// TIA Portal V15.1 export
// export: Created 2024-06-21T08:41:07.0870984Z, ExportSetting WithDefaults, DisplayName Totally Integrated Automation Portal, DisplayVersion V15.1 Update 5, DisplayName TIA Portal Openness, DisplayVersion V15.1 Update 5, DisplayName SINAMICS Startdrive Advanced, DisplayVersion V15.1, DisplayName G130, G150, S120, S150, SINAMICS MV, S210, DisplayVersion V15.1, DisplayName G110M, G120, G120C, G120D, G120P, DisplayVersion V15.1, DisplayName STEP 7 Professional, DisplayVersion V15.1 Update 5, DisplayName STEP 7 Safety, DisplayVersion V15.1, DisplayName WinCC Professional, DisplayVersion V15.1 Update 5, DisplayName SIMATIC Visualization Architect, DisplayVersion V15.1
FUNCTION_BLOCK "LGBBodyCounter"   // FB6602, FBD
TITLE = Body Counter Dynamic
{ S7_Optimized_Access := 'TRUE' }
AUTHOR : CSTAAL
VERSION : 0.1
// stored: AutoNumber false, IsIECCheckEnabled false, IsRetainMemResEnabled false, MemoryReserve 100, SetENOAutomatically False, UDAEnableTagReadback false
   VAR_INPUT
      I_EnableDynamicMax { ExternalAccessible := 'False'; ExternalVisible := 'False'; ExternalWritable := 'False'} : Bool;   // Dynamic Maximum Enabled
      I_MaxBody { ExternalAccessible := 'False'; ExternalVisible := 'False'; ExternalWritable := 'False'} : DInt;   // Max Amount of Bodies in the Zone
      I_DPBody { ExternalAccessible := 'False'; ExternalVisible := 'False'; ExternalWritable := 'False'} : Bool;   // DP Body Type Used in Zone
      I_ECBody { ExternalAccessible := 'False'; ExternalVisible := 'False'; ExternalWritable := 'False'} : Bool;   // EC Body Type Used in Zone
      I_ECSkid { ExternalAccessible := 'False'; ExternalVisible := 'False'; ExternalWritable := 'False'} : Bool;   // EC Skid Type Used in Zone
      I_PaintedBody { ExternalAccessible := 'False'; ExternalVisible := 'False'; ExternalWritable := 'False'} : Bool;   // Painted Body Type Used in Zone
      I_Conv1Enable { ExternalAccessible := 'False'; ExternalVisible := 'False'; ExternalWritable := 'False'} : Bool;   // Enable Conveyor 1
      I_Conv1MaxBody { ExternalAccessible := 'False'; ExternalVisible := 'False'; ExternalWritable := 'False'} : DInt;   // Max Amount of Bodies on Conveyor 1
      I_Conv1SetTrfInTrf { ExternalAccessible := 'False'; ExternalVisible := 'False'; ExternalWritable := 'False'} : Bool;   // Transfer In Set Conveyor 1
      I_Conv1SetTrfOutTrf { ExternalAccessible := 'False'; ExternalVisible := 'False'; ExternalWritable := 'False'} : Bool;   // Transfer Out Set Conveyor 1
      I_Conv1ResTrfInTrf { ExternalAccessible := 'False'; ExternalVisible := 'False'; ExternalWritable := 'False'} : Bool;   // Transfer In Reset Conveyor 1
      I_Conv1ResTrfOutTrf { ExternalAccessible := 'False'; ExternalVisible := 'False'; ExternalWritable := 'False'} : Bool;   // Transfer Out Reset Conveyor 1
      I_Conv2Enable { ExternalAccessible := 'False'; ExternalVisible := 'False'; ExternalWritable := 'False'} : Bool;   // Enable Conveyor 2
      I_Conv2MaxBody { ExternalAccessible := 'False'; ExternalVisible := 'False'; ExternalWritable := 'False'} : DInt;   // Max Amount of Bodies on Conveyor 2
      I_Conv2SetTrfInTrf { ExternalAccessible := 'False'; ExternalVisible := 'False'; ExternalWritable := 'False'} : Bool;   // Transfer In Set Conveyor 2
      I_Conv2SetTrfOutTrf { ExternalAccessible := 'False'; ExternalVisible := 'False'; ExternalWritable := 'False'} : Bool;   // Transfer Out Set Conveyor 2
      I_Conv2ResTrfInTrf { ExternalAccessible := 'False'; ExternalVisible := 'False'; ExternalWritable := 'False'} : Bool;   // Transfer In Reset Conveyor 2
      I_Conv2ResTrfOutTrf { ExternalAccessible := 'False'; ExternalVisible := 'False'; ExternalWritable := 'False'} : Bool;   // Transfer Out Reset Conveyor 2
      I_Pos1BodyPresent { ExternalAccessible := 'False'; ExternalVisible := 'False'; ExternalWritable := 'False'} : Bool;   // Position 1 Body Present
      I_Pos1RollerSetInTrf { ExternalAccessible := 'False'; ExternalVisible := 'False'; ExternalWritable := 'False'} : Bool;   // Position 1 Roller Transfer In Set
      I_Pos1RollerResInTrf { ExternalAccessible := 'False'; ExternalVisible := 'False'; ExternalWritable := 'False'} : Bool;   // Position 1 Roller Transfer In Reset
      I_Pos1CCSetInTrf { ExternalAccessible := 'False'; ExternalVisible := 'False'; ExternalWritable := 'False'} : Bool;   // Position 1 Cross Conveyor Transfer In Set
      I_Pos1CCResInTrf { ExternalAccessible := 'False'; ExternalVisible := 'False'; ExternalWritable := 'False'} : Bool;   // Position 1 Cross Conveyor Transfer In Reset
      I_Pos1RollerSetOutTrf { ExternalAccessible := 'False'; ExternalVisible := 'False'; ExternalWritable := 'False'} : Bool;   // Position 1 Roller Transfer Out Set
      I_Pos1RollerResOutTrf { ExternalAccessible := 'False'; ExternalVisible := 'False'; ExternalWritable := 'False'} : Bool;   // Position 1 Roller Transfer Out Reset
      I_Pos1CCSetOutTrf { ExternalAccessible := 'False'; ExternalVisible := 'False'; ExternalWritable := 'False'} : Bool;   // Position 1 Cross Conveyor Transfer Out Set
      I_Pos1CCResOutTrf { ExternalAccessible := 'False'; ExternalVisible := 'False'; ExternalWritable := 'False'} : Bool;   // Position 1 Cross Conveyor Transfer Out Reset
      I_Pos2BodyPresent { ExternalAccessible := 'False'; ExternalVisible := 'False'; ExternalWritable := 'False'} : Bool;   // Position 2 Body Present
      I_Pos2RollerSetInTrf { ExternalAccessible := 'False'; ExternalVisible := 'False'; ExternalWritable := 'False'} : Bool;   // Position 2 Roller Transfer In Set
      I_Pos2RollerResInTrf { ExternalAccessible := 'False'; ExternalVisible := 'False'; ExternalWritable := 'False'} : Bool;   // Position 2 Roller Transfer In Reset
      I_Pos2CCSetInTrf { ExternalAccessible := 'False'; ExternalVisible := 'False'; ExternalWritable := 'False'} : Bool;   // Position 2 Cross Conveyor Transfer In Set
      I_Pos2CCResInTrf { ExternalAccessible := 'False'; ExternalVisible := 'False'; ExternalWritable := 'False'} : Bool;   // Position 2 Cross Conveyor Transfer In Reset
      I_Pos2RollerSetOutTrf { ExternalAccessible := 'False'; ExternalVisible := 'False'; ExternalWritable := 'False'} : Bool;   // Position 2 Roller Transfer Out Set
      I_Pos2RollerResOutTrf { ExternalAccessible := 'False'; ExternalVisible := 'False'; ExternalWritable := 'False'} : Bool;   // Position 2 Roller Transfer Out Reset
      I_Pos2CCSetOutTrf { ExternalAccessible := 'False'; ExternalVisible := 'False'; ExternalWritable := 'False'} : Bool;   // Position 2 Cross Conveyor Transfer Out Set
      I_Pos2CCResOutTrf { ExternalAccessible := 'False'; ExternalVisible := 'False'; ExternalWritable := 'False'} : Bool;   // Position 2 Cross Conveyor Transfer Out Reset
      I_Pos3BodyPresent { ExternalAccessible := 'False'; ExternalVisible := 'False'; ExternalWritable := 'False'} : Bool;   // Position 3 Body Present
      I_Pos3RollerSetInTrf { ExternalAccessible := 'False'; ExternalVisible := 'False'; ExternalWritable := 'False'} : Bool;   // Position 3 Roller Transfer In Set
      I_Pos3RollerResInTrf { ExternalAccessible := 'False'; ExternalVisible := 'False'; ExternalWritable := 'False'} : Bool;   // Position 3 Roller Transfer In Reset
      I_Pos3CCSetInTrf { ExternalAccessible := 'False'; ExternalVisible := 'False'; ExternalWritable := 'False'} : Bool;   // Position 3 Cross Conveyor Transfer In Set
      I_Pos3CCResInTrf { ExternalAccessible := 'False'; ExternalVisible := 'False'; ExternalWritable := 'False'} : Bool;   // Position 3 Cross Conveyor Transfer In Reset
      I_Pos3RollerSetOutTrf { ExternalAccessible := 'False'; ExternalVisible := 'False'; ExternalWritable := 'False'} : Bool;   // Position 3 Roller Transfer Out Set
      I_Pos3RollerResOutTrf { ExternalAccessible := 'False'; ExternalVisible := 'False'; ExternalWritable := 'False'} : Bool;   // Position 3 Roller Transfer Out Reset
      I_Pos3CCSetOutTrf { ExternalAccessible := 'False'; ExternalVisible := 'False'; ExternalWritable := 'False'} : Bool;   // Position 3 Cross Conveyor Transfer Out Set
      I_Pos3CCResOutTrf { ExternalAccessible := 'False'; ExternalVisible := 'False'; ExternalWritable := 'False'} : Bool;   // Position 3 Cross Conveyor Transfer Out Reset
      I_Pos4BodyPresent { ExternalAccessible := 'False'; ExternalVisible := 'False'; ExternalWritable := 'False'} : Bool;   // Position 4 Body Present
      I_Pos4RollerSetInTrf { ExternalAccessible := 'False'; ExternalVisible := 'False'; ExternalWritable := 'False'} : Bool;   // Position 4 Roller Transfer In Set
      I_Pos4RollerResInTrf { ExternalAccessible := 'False'; ExternalVisible := 'False'; ExternalWritable := 'False'} : Bool;   // Position 4 Roller Transfer In Reset
      I_Pos4CCSetInTrf { ExternalAccessible := 'False'; ExternalVisible := 'False'; ExternalWritable := 'False'} : Bool;   // Position 4 Cross Conveyor Transfer In Set
      I_Pos4CCResInTrf { ExternalAccessible := 'False'; ExternalVisible := 'False'; ExternalWritable := 'False'} : Bool;   // Position 4 Cross Conveyor Transfer In Reset
      I_Pos4RollerSetOutTrf { ExternalAccessible := 'False'; ExternalVisible := 'False'; ExternalWritable := 'False'} : Bool;   // Position 4 Roller Transfer Out Set
      I_Pos4RollerResOutTrf { ExternalAccessible := 'False'; ExternalVisible := 'False'; ExternalWritable := 'False'} : Bool;   // Position 4 Roller Transfer Out Reset
      I_Pos4CCSetOutTrf { ExternalAccessible := 'False'; ExternalVisible := 'False'; ExternalWritable := 'False'} : Bool;   // Position 4 Cross Conveyor Transfer Out Set
      I_Pos4CCResOutTrf { ExternalAccessible := 'False'; ExternalVisible := 'False'; ExternalWritable := 'False'} : Bool;   // Position 4 Cross Conveyor Transfer Out Reset
      I_Pos5BodyPresent { ExternalAccessible := 'False'; ExternalVisible := 'False'; ExternalWritable := 'False'} : Bool;   // Position 5 Body Present
      I_Pos5RollerSetInTrf { ExternalAccessible := 'False'; ExternalVisible := 'False'; ExternalWritable := 'False'} : Bool;   // Position 5 Roller Transfer In Set
      I_Pos5RollerResInTrf { ExternalAccessible := 'False'; ExternalVisible := 'False'; ExternalWritable := 'False'} : Bool;   // Position 5 Roller Transfer In Reset
      I_Pos5CCSetInTrf { ExternalAccessible := 'False'; ExternalVisible := 'False'; ExternalWritable := 'False'} : Bool;   // Position 5 Cross Conveyor Transfer In Set
      I_Pos5CCResInTrf { ExternalAccessible := 'False'; ExternalVisible := 'False'; ExternalWritable := 'False'} : Bool;   // Position 5 Cross Conveyor Transfer In Reset
      I_Pos5RollerSetOutTrf { ExternalAccessible := 'False'; ExternalVisible := 'False'; ExternalWritable := 'False'} : Bool;   // Position 5 Roller Transfer Out Set
      I_Pos5RollerResOutTrf { ExternalAccessible := 'False'; ExternalVisible := 'False'; ExternalWritable := 'False'} : Bool;   // Position 5 Roller Transfer Out Reset
      I_Pos5CCSetOutTrf { ExternalAccessible := 'False'; ExternalVisible := 'False'; ExternalWritable := 'False'} : Bool;   // Position 5 Cross Conveyor Transfer Out Set
      I_Pos5CCResOutTrf { ExternalAccessible := 'False'; ExternalVisible := 'False'; ExternalWritable := 'False'} : Bool;   // Position 5 Cross Conveyor Transfer Out Reset
      I_Pos6BodyPresent { ExternalAccessible := 'False'; ExternalVisible := 'False'; ExternalWritable := 'False'} : Bool;   // Position 6 Body Present
      I_Pos6RollerSetInTrf { ExternalAccessible := 'False'; ExternalVisible := 'False'; ExternalWritable := 'False'} : Bool;   // Position 6 Roller Transfer In Set
      I_Pos6RollerResInTrf { ExternalAccessible := 'False'; ExternalVisible := 'False'; ExternalWritable := 'False'} : Bool;   // Position 6 Roller Transfer In Reset
      I_Pos6CCSetInTrf { ExternalAccessible := 'False'; ExternalVisible := 'False'; ExternalWritable := 'False'} : Bool;   // Position 6 Cross Conveyor Transfer In Set
      I_Pos6CCResInTrf { ExternalAccessible := 'False'; ExternalVisible := 'False'; ExternalWritable := 'False'} : Bool;   // Position 6 Cross Conveyor Transfer In Reset
      I_Pos6RollerSetOutTrf { ExternalAccessible := 'False'; ExternalVisible := 'False'; ExternalWritable := 'False'} : Bool;   // Position 6 Roller Transfer Out Set
      I_Pos6RollerResOutTrf { ExternalAccessible := 'False'; ExternalVisible := 'False'; ExternalWritable := 'False'} : Bool;   // Position 6 Roller Transfer Out Reset
      I_Pos6CCSetOutTrf { ExternalAccessible := 'False'; ExternalVisible := 'False'; ExternalWritable := 'False'} : Bool;   // Position 6 Cross Conveyor Transfer Out Set
      I_Pos6CCResOutTrf { ExternalAccessible := 'False'; ExternalVisible := 'False'; ExternalWritable := 'False'} : Bool;   // Position 6 Cross Conveyor Transfer Out Reset
      I_Pos7BodyPresent { ExternalAccessible := 'False'; ExternalVisible := 'False'; ExternalWritable := 'False'} : Bool;   // Position 7 Body Present
      I_Pos7RollerSetInTrf { ExternalAccessible := 'False'; ExternalVisible := 'False'; ExternalWritable := 'False'} : Bool;   // Position 7 Roller Transfer In Set
      I_Pos7RollerResInTrf { ExternalAccessible := 'False'; ExternalVisible := 'False'; ExternalWritable := 'False'} : Bool;   // Position 7 Roller Transfer In Reset
      I_Pos7CCSetInTrf { ExternalAccessible := 'False'; ExternalVisible := 'False'; ExternalWritable := 'False'} : Bool;   // Position 7 Cross Conveyor Transfer In Set
      I_Pos7CCResInTrf { ExternalAccessible := 'False'; ExternalVisible := 'False'; ExternalWritable := 'False'} : Bool;   // Position 7 Cross Conveyor Transfer In Reset
      I_Pos7RollerSetOutTrf { ExternalAccessible := 'False'; ExternalVisible := 'False'; ExternalWritable := 'False'} : Bool;   // Position 7 Roller Transfer Out Set
      I_Pos7RollerResOutTrf { ExternalAccessible := 'False'; ExternalVisible := 'False'; ExternalWritable := 'False'} : Bool;   // Position 7 Roller Transfer Out Reset
      I_Pos7CCSetOutTrf { ExternalAccessible := 'False'; ExternalVisible := 'False'; ExternalWritable := 'False'} : Bool;   // Position 7 Cross Conveyor Transfer Out Set
      I_Pos7CCResOutTrf { ExternalAccessible := 'False'; ExternalVisible := 'False'; ExternalWritable := 'False'} : Bool;   // Position 7 Cross Conveyor Transfer Out Reset
      I_Pos8BodyPresent { ExternalAccessible := 'False'; ExternalVisible := 'False'; ExternalWritable := 'False'} : Bool;   // Position 8 Body Present
      I_Pos8RollerSetInTrf { ExternalAccessible := 'False'; ExternalVisible := 'False'; ExternalWritable := 'False'} : Bool;   // Position 8 Roller Transfer In Set
      I_Pos8RollerResInTrf { ExternalAccessible := 'False'; ExternalVisible := 'False'; ExternalWritable := 'False'} : Bool;   // Position 8 Roller Transfer In Reset
      I_Pos8CCSetInTrf { ExternalAccessible := 'False'; ExternalVisible := 'False'; ExternalWritable := 'False'} : Bool;   // Position 8 Cross Conveyor Transfer In Set
      I_Pos8CCResInTrf { ExternalAccessible := 'False'; ExternalVisible := 'False'; ExternalWritable := 'False'} : Bool;   // Position 8 Cross Conveyor Transfer In Reset
      I_Pos8RollerSetOutTrf { ExternalAccessible := 'False'; ExternalVisible := 'False'; ExternalWritable := 'False'} : Bool;   // Position 8 Roller Transfer Out Set
      I_Pos8RollerResOutTrf { ExternalAccessible := 'False'; ExternalVisible := 'False'; ExternalWritable := 'False'} : Bool;   // Position 8 Roller Transfer Out Reset
      I_Pos8CCSetOutTrf { ExternalAccessible := 'False'; ExternalVisible := 'False'; ExternalWritable := 'False'} : Bool;   // Position 8 Cross Conveyor Transfer Out Set
      I_Pos8CCResOutTrf { ExternalAccessible := 'False'; ExternalVisible := 'False'; ExternalWritable := 'False'} : Bool;   // Position 8 Cross Conveyor Transfer Out Reset
      I_Pos9BodyPresent { ExternalAccessible := 'False'; ExternalVisible := 'False'; ExternalWritable := 'False'} : Bool;   // Position 9 Body Present
      I_Pos9RollerSetInTrf { ExternalAccessible := 'False'; ExternalVisible := 'False'; ExternalWritable := 'False'} : Bool;   // Position 9 Roller Transfer In Set
      I_Pos9RollerResInTrf { ExternalAccessible := 'False'; ExternalVisible := 'False'; ExternalWritable := 'False'} : Bool;   // Position 9 Roller Transfer In Reset
      I_Pos9CCSetInTrf { ExternalAccessible := 'False'; ExternalVisible := 'False'; ExternalWritable := 'False'} : Bool;   // Position 9 Cross Conveyor Transfer In Set
      I_Pos9CCResInTrf { ExternalAccessible := 'False'; ExternalVisible := 'False'; ExternalWritable := 'False'} : Bool;   // Position 9 Cross Conveyor Transfer In Reset
      I_Pos9RollerSetOutTrf { ExternalAccessible := 'False'; ExternalVisible := 'False'; ExternalWritable := 'False'} : Bool;   // Position 9 Roller Transfer Out Set
      I_Pos9RollerResOutTrf { ExternalAccessible := 'False'; ExternalVisible := 'False'; ExternalWritable := 'False'} : Bool;   // Position 9 Roller Transfer Out Reset
      I_Pos9CCSetOutTrf { ExternalAccessible := 'False'; ExternalVisible := 'False'; ExternalWritable := 'False'} : Bool;   // Position 9 Cross Conveyor Transfer Out Set
      I_Pos9CCResOutTrf { ExternalAccessible := 'False'; ExternalVisible := 'False'; ExternalWritable := 'False'} : Bool;   // Position 9 Cross Conveyor Transfer Out Reset
      I_Pos10BodyPresent { ExternalAccessible := 'False'; ExternalVisible := 'False'; ExternalWritable := 'False'} : Bool;   // Position 10 Body Present
      I_Pos10RollerSetInTrf { ExternalAccessible := 'False'; ExternalVisible := 'False'; ExternalWritable := 'False'} : Bool;   // Position 10 Roller Transfer In Set
      I_Pos10RollerResInTrf { ExternalAccessible := 'False'; ExternalVisible := 'False'; ExternalWritable := 'False'} : Bool;   // Position 10 Roller Transfer In Reset
      I_Pos10CCSetInTrf { ExternalAccessible := 'False'; ExternalVisible := 'False'; ExternalWritable := 'False'} : Bool;   // Position 10 Cross Conveyor Transfer In Set
      I_Pos10CCResInTrf { ExternalAccessible := 'False'; ExternalVisible := 'False'; ExternalWritable := 'False'} : Bool;   // Position 10 Cross Conveyor Transfer In Reset
      I_Pos10RollerSetOutTrf { ExternalAccessible := 'False'; ExternalVisible := 'False'; ExternalWritable := 'False'} : Bool;   // Position 10 Roller Transfer Out Set
      I_Pos10RollerResOutTrf { ExternalAccessible := 'False'; ExternalVisible := 'False'; ExternalWritable := 'False'} : Bool;   // Position 10 Roller Transfer Out Reset
      I_Pos10CCSetOutTrf { ExternalAccessible := 'False'; ExternalVisible := 'False'; ExternalWritable := 'False'} : Bool;   // Position 10 Cross Conveyor Transfer Out Set
      I_Pos10CCResOutTrf { ExternalAccessible := 'False'; ExternalVisible := 'False'; ExternalWritable := 'False'} : Bool;   // Position 10 Cross Conveyor Transfer Out Reset
      I_Pos11BodyPresent { ExternalAccessible := 'False'; ExternalVisible := 'False'; ExternalWritable := 'False'} : Bool;   // Position 11 Body Present
      I_Pos11RollerSetInTrf { ExternalAccessible := 'False'; ExternalVisible := 'False'; ExternalWritable := 'False'} : Bool;   // Position 11 Roller Transfer In Set
      I_Pos11RollerResInTrf { ExternalAccessible := 'False'; ExternalVisible := 'False'; ExternalWritable := 'False'} : Bool;   // Position 11 Roller Transfer In Reset
      I_Pos11CCSetInTrf { ExternalAccessible := 'False'; ExternalVisible := 'False'; ExternalWritable := 'False'} : Bool;   // Position 11 Cross Conveyor Transfer In Set
      I_Pos11CCResInTrf { ExternalAccessible := 'False'; ExternalVisible := 'False'; ExternalWritable := 'False'} : Bool;   // Position 11 Cross Conveyor Transfer In Reset
      I_Pos11RollerSetOutTrf { ExternalAccessible := 'False'; ExternalVisible := 'False'; ExternalWritable := 'False'} : Bool;   // Position 11 Roller Transfer Out Set
      I_Pos11RollerResOutTrf { ExternalAccessible := 'False'; ExternalVisible := 'False'; ExternalWritable := 'False'} : Bool;   // Position 11 Roller Transfer Out Reset
      I_Pos11CCSetOutTrf { ExternalAccessible := 'False'; ExternalVisible := 'False'; ExternalWritable := 'False'} : Bool;   // Position 11 Cross Conveyor Transfer Out Set
      I_Pos11CCResOutTrf { ExternalAccessible := 'False'; ExternalVisible := 'False'; ExternalWritable := 'False'} : Bool;   // Position 11 Cross Conveyor Transfer Out Reset
      I_Pos12BodyPresent { ExternalAccessible := 'False'; ExternalVisible := 'False'; ExternalWritable := 'False'} : Bool;   // Position 12 Body Present
      I_Pos12RollerSetInTrf { ExternalAccessible := 'False'; ExternalVisible := 'False'; ExternalWritable := 'False'} : Bool;   // Position 12 Roller Transfer In Set
      I_Pos12RollerResInTrf { ExternalAccessible := 'False'; ExternalVisible := 'False'; ExternalWritable := 'False'} : Bool;   // Position 12 Roller Transfer In Reset
      I_Pos12CCSetInTrf { ExternalAccessible := 'False'; ExternalVisible := 'False'; ExternalWritable := 'False'} : Bool;   // Position 12 Cross Conveyor Transfer In Set
      I_Pos12CCResInTrf { ExternalAccessible := 'False'; ExternalVisible := 'False'; ExternalWritable := 'False'} : Bool;   // Position 12 Cross Conveyor Transfer In Reset
      I_Pos12RollerSetOutTrf { ExternalAccessible := 'False'; ExternalVisible := 'False'; ExternalWritable := 'False'} : Bool;   // Position 12 Roller Transfer Out Set
      I_Pos12RollerResOutTrf { ExternalAccessible := 'False'; ExternalVisible := 'False'; ExternalWritable := 'False'} : Bool;   // Position 12 Roller Transfer Out Reset
      I_Pos12CCSetOutTrf { ExternalAccessible := 'False'; ExternalVisible := 'False'; ExternalWritable := 'False'} : Bool;   // Position 12 Cross Conveyor Transfer Out Set
      I_Pos12CCResOutTrf { ExternalAccessible := 'False'; ExternalVisible := 'False'; ExternalWritable := 'False'} : Bool;   // Position 12 Cross Conveyor Transfer Out Reset
      I_Pos13BodyPresent { ExternalAccessible := 'False'; ExternalVisible := 'False'; ExternalWritable := 'False'} : Bool;   // Position 13 Body Present
      I_Pos13RollerSetInTrf { ExternalAccessible := 'False'; ExternalVisible := 'False'; ExternalWritable := 'False'} : Bool;   // Position 13 Roller Transfer In Set
      I_Pos13RollerResInTrf { ExternalAccessible := 'False'; ExternalVisible := 'False'; ExternalWritable := 'False'} : Bool;   // Position 13 Roller Transfer In Reset
      I_Pos13CCSetInTrf { ExternalAccessible := 'False'; ExternalVisible := 'False'; ExternalWritable := 'False'} : Bool;   // Position 13 Cross Conveyor Transfer In Set
      I_Pos13CCResInTrf { ExternalAccessible := 'False'; ExternalVisible := 'False'; ExternalWritable := 'False'} : Bool;   // Position 13 Cross Conveyor Transfer In Reset
      I_Pos13RollerSetOutTrf { ExternalAccessible := 'False'; ExternalVisible := 'False'; ExternalWritable := 'False'} : Bool;   // Position 13 Roller Transfer Out Set
      I_Pos13RollerResOutTrf { ExternalAccessible := 'False'; ExternalVisible := 'False'; ExternalWritable := 'False'} : Bool;   // Position 13 Roller Transfer Out Reset
      I_Pos13CCSetOutTrf { ExternalAccessible := 'False'; ExternalVisible := 'False'; ExternalWritable := 'False'} : Bool;   // Position 13 Cross Conveyor Transfer Out Set
      I_Pos13CCResOutTrf { ExternalAccessible := 'False'; ExternalVisible := 'False'; ExternalWritable := 'False'} : Bool;   // Position 13 Cross Conveyor Transfer Out Reset
      I_Pos14BodyPresent { ExternalAccessible := 'False'; ExternalVisible := 'False'; ExternalWritable := 'False'} : Bool;   // Position 14 Body Present
      I_Pos14RollerSetInTrf { ExternalAccessible := 'False'; ExternalVisible := 'False'; ExternalWritable := 'False'} : Bool;   // Position 14 Roller Transfer In Set
      I_Pos14RollerResInTrf { ExternalAccessible := 'False'; ExternalVisible := 'False'; ExternalWritable := 'False'} : Bool;   // Position 14 Roller Transfer In Reset
      I_Pos14CCSetInTrf { ExternalAccessible := 'False'; ExternalVisible := 'False'; ExternalWritable := 'False'} : Bool;   // Position 14 Cross Conveyor Transfer In Set
      I_Pos14CCResInTrf { ExternalAccessible := 'False'; ExternalVisible := 'False'; ExternalWritable := 'False'} : Bool;   // Position 14 Cross Conveyor Transfer In Reset
      I_Pos14RollerSetOutTrf { ExternalAccessible := 'False'; ExternalVisible := 'False'; ExternalWritable := 'False'} : Bool;   // Position 14 Roller Transfer Out Set
      I_Pos14RollerResOutTrf { ExternalAccessible := 'False'; ExternalVisible := 'False'; ExternalWritable := 'False'} : Bool;   // Position 14 Roller Transfer Out Reset
      I_Pos14CCSetOutTrf { ExternalAccessible := 'False'; ExternalVisible := 'False'; ExternalWritable := 'False'} : Bool;   // Position 14 Cross Conveyor Transfer Out Set
      I_Pos14CCResOutTrf { ExternalAccessible := 'False'; ExternalVisible := 'False'; ExternalWritable := 'False'} : Bool;   // Position 14 Cross Conveyor Transfer Out Reset
      I_Pos15BodyPresent { ExternalAccessible := 'False'; ExternalVisible := 'False'; ExternalWritable := 'False'} : Bool;   // Position 15 Body Present
      I_Pos15RollerSetInTrf { ExternalAccessible := 'False'; ExternalVisible := 'False'; ExternalWritable := 'False'} : Bool;   // Position 15 Roller Transfer In Set
      I_Pos15RollerResInTrf { ExternalAccessible := 'False'; ExternalVisible := 'False'; ExternalWritable := 'False'} : Bool;   // Position 15 Roller Transfer In Reset
      I_Pos15CCSetInTrf { ExternalAccessible := 'False'; ExternalVisible := 'False'; ExternalWritable := 'False'} : Bool;   // Position 15 Cross Conveyor Transfer In Set
      I_Pos15CCResInTrf { ExternalAccessible := 'False'; ExternalVisible := 'False'; ExternalWritable := 'False'} : Bool;   // Position 15 Cross Conveyor Transfer In Reset
      I_Pos15RollerSetOutTrf { ExternalAccessible := 'False'; ExternalVisible := 'False'; ExternalWritable := 'False'} : Bool;   // Position 15 Roller Transfer Out Set
      I_Pos15RollerResOutTrf { ExternalAccessible := 'False'; ExternalVisible := 'False'; ExternalWritable := 'False'} : Bool;   // Position 15 Roller Transfer Out Reset
      I_Pos15CCSetOutTrf { ExternalAccessible := 'False'; ExternalVisible := 'False'; ExternalWritable := 'False'} : Bool;   // Position 15 Cross Conveyor Transfer Out Set
      I_Pos15CCResOutTrf { ExternalAccessible := 'False'; ExternalVisible := 'False'; ExternalWritable := 'False'} : Bool;   // Position 15 Cross Conveyor Transfer Out Reset
      I_Pos16BodyPresent { ExternalAccessible := 'False'; ExternalVisible := 'False'; ExternalWritable := 'False'} : Bool;   // Position 16 Body Present
      I_Pos16RollerSetInTrf { ExternalAccessible := 'False'; ExternalVisible := 'False'; ExternalWritable := 'False'} : Bool;   // Position 16 Roller Transfer In Set
      I_Pos16RollerResInTrf { ExternalAccessible := 'False'; ExternalVisible := 'False'; ExternalWritable := 'False'} : Bool;   // Position 16 Roller Transfer In Reset
      I_Pos16CCSetInTrf { ExternalAccessible := 'False'; ExternalVisible := 'False'; ExternalWritable := 'False'} : Bool;   // Position 16 Cross Conveyor Transfer In Set
      I_Pos16CCResInTrf { ExternalAccessible := 'False'; ExternalVisible := 'False'; ExternalWritable := 'False'} : Bool;   // Position 16 Cross Conveyor Transfer In Reset
      I_Pos16RollerSetOutTrf { ExternalAccessible := 'False'; ExternalVisible := 'False'; ExternalWritable := 'False'} : Bool;   // Position 16 Roller Transfer Out Set
      I_Pos16RollerResOutTrf { ExternalAccessible := 'False'; ExternalVisible := 'False'; ExternalWritable := 'False'} : Bool;   // Position 16 Roller Transfer Out Reset
      I_Pos16CCSetOutTrf { ExternalAccessible := 'False'; ExternalVisible := 'False'; ExternalWritable := 'False'} : Bool;   // Position 16 Cross Conveyor Transfer Out Set
      I_Pos16CCResOutTrf { ExternalAccessible := 'False'; ExternalVisible := 'False'; ExternalWritable := 'False'} : Bool;   // Position 16 Cross Conveyor Transfer Out Reset
      I_Pos17BodyPresent { ExternalAccessible := 'False'; ExternalVisible := 'False'; ExternalWritable := 'False'} : Bool;   // Position 17 Body Present
      I_Pos17RollerSetInTrf { ExternalAccessible := 'False'; ExternalVisible := 'False'; ExternalWritable := 'False'} : Bool;   // Position 17 Roller Transfer In Set
      I_Pos17RollerResInTrf { ExternalAccessible := 'False'; ExternalVisible := 'False'; ExternalWritable := 'False'} : Bool;   // Position 17 Roller Transfer In Reset
      I_Pos17CCSetInTrf { ExternalAccessible := 'False'; ExternalVisible := 'False'; ExternalWritable := 'False'} : Bool;   // Position 17 Cross Conveyor Transfer In Set
      I_Pos17CCResInTrf { ExternalAccessible := 'False'; ExternalVisible := 'False'; ExternalWritable := 'False'} : Bool;   // Position 17 Cross Conveyor Transfer In Reset
      I_Pos17RollerSetOutTrf { ExternalAccessible := 'False'; ExternalVisible := 'False'; ExternalWritable := 'False'} : Bool;   // Position 17 Roller Transfer Out Set
      I_Pos17RollerResOutTrf { ExternalAccessible := 'False'; ExternalVisible := 'False'; ExternalWritable := 'False'} : Bool;   // Position 17 Roller Transfer Out Reset
      I_Pos17CCSetOutTrf { ExternalAccessible := 'False'; ExternalVisible := 'False'; ExternalWritable := 'False'} : Bool;   // Position 17 Cross Conveyor Transfer Out Set
      I_Pos17CCResOutTrf { ExternalAccessible := 'False'; ExternalVisible := 'False'; ExternalWritable := 'False'} : Bool;   // Position 17 Cross Conveyor Transfer Out Reset
      I_Pos18BodyPresent { ExternalAccessible := 'False'; ExternalVisible := 'False'; ExternalWritable := 'False'} : Bool;   // Position 18 Body Present
      I_Pos18RollerSetInTrf { ExternalAccessible := 'False'; ExternalVisible := 'False'; ExternalWritable := 'False'} : Bool;   // Position 18 Roller Transfer In Set
      I_Pos18RollerResInTrf { ExternalAccessible := 'False'; ExternalVisible := 'False'; ExternalWritable := 'False'} : Bool;   // Position 18 Roller Transfer In Reset
      I_Pos18CCSetInTrf { ExternalAccessible := 'False'; ExternalVisible := 'False'; ExternalWritable := 'False'} : Bool;   // Position 18 Cross Conveyor Transfer In Set
      I_Pos18CCResInTrf { ExternalAccessible := 'False'; ExternalVisible := 'False'; ExternalWritable := 'False'} : Bool;   // Position 18 Cross Conveyor Transfer In Reset
      I_Pos18RollerSetOutTrf { ExternalAccessible := 'False'; ExternalVisible := 'False'; ExternalWritable := 'False'} : Bool;   // Position 18 Roller Transfer Out Set
      I_Pos18RollerResOutTrf { ExternalAccessible := 'False'; ExternalVisible := 'False'; ExternalWritable := 'False'} : Bool;   // Position 18 Roller Transfer Out Reset
      I_Pos18CCSetOutTrf { ExternalAccessible := 'False'; ExternalVisible := 'False'; ExternalWritable := 'False'} : Bool;   // Position 18 Cross Conveyor Transfer Out Set
      I_Pos18CCResOutTrf { ExternalAccessible := 'False'; ExternalVisible := 'False'; ExternalWritable := 'False'} : Bool;   // Position 18 Cross Conveyor Transfer Out Reset
      I_Pos19BodyPresent { ExternalAccessible := 'False'; ExternalVisible := 'False'; ExternalWritable := 'False'} : Bool;   // Position 19 Body Present
      I_Pos19RollerSetInTrf { ExternalAccessible := 'False'; ExternalVisible := 'False'; ExternalWritable := 'False'} : Bool;   // Position 19 Roller Transfer In Set
      I_Pos19RollerResInTrf { ExternalAccessible := 'False'; ExternalVisible := 'False'; ExternalWritable := 'False'} : Bool;   // Position 19 Roller Transfer In Reset
      I_Pos19CCSetInTrf { ExternalAccessible := 'False'; ExternalVisible := 'False'; ExternalWritable := 'False'} : Bool;   // Position 19 Cross Conveyor Transfer In Set
      I_Pos19CCResInTrf { ExternalAccessible := 'False'; ExternalVisible := 'False'; ExternalWritable := 'False'} : Bool;   // Position 19 Cross Conveyor Transfer In Reset
      I_Pos19RollerSetOutTrf { ExternalAccessible := 'False'; ExternalVisible := 'False'; ExternalWritable := 'False'} : Bool;   // Position 19 Roller Transfer Out Set
      I_Pos19RollerResOutTrf { ExternalAccessible := 'False'; ExternalVisible := 'False'; ExternalWritable := 'False'} : Bool;   // Position 19 Roller Transfer Out Reset
      I_Pos19CCSetOutTrf { ExternalAccessible := 'False'; ExternalVisible := 'False'; ExternalWritable := 'False'} : Bool;   // Position 19 Cross Conveyor Transfer Out Set
      I_Pos19CCResOutTrf { ExternalAccessible := 'False'; ExternalVisible := 'False'; ExternalWritable := 'False'} : Bool;   // Position 19 Cross Conveyor Transfer Out Reset
      I_Pos20BodyPresent { ExternalAccessible := 'False'; ExternalVisible := 'False'; ExternalWritable := 'False'} : Bool;   // Position 20 Body Present
      I_Pos20RollerSetInTrf { ExternalAccessible := 'False'; ExternalVisible := 'False'; ExternalWritable := 'False'} : Bool;   // Position 20 Roller Transfer In Set
      I_Pos20RollerResInTrf { ExternalAccessible := 'False'; ExternalVisible := 'False'; ExternalWritable := 'False'} : Bool;   // Position 20 Roller Transfer In Reset
      I_Pos20CCSetInTrf { ExternalAccessible := 'False'; ExternalVisible := 'False'; ExternalWritable := 'False'} : Bool;   // Position 20 Cross Conveyor Transfer In Set
      I_Pos20CCResInTrf { ExternalAccessible := 'False'; ExternalVisible := 'False'; ExternalWritable := 'False'} : Bool;   // Position 20 Cross Conveyor Transfer In Reset
      I_Pos20RollerSetOutTrf { ExternalAccessible := 'False'; ExternalVisible := 'False'; ExternalWritable := 'False'} : Bool;   // Position 20 Roller Transfer Out Set
      I_Pos20RollerResOutTrf { ExternalAccessible := 'False'; ExternalVisible := 'False'; ExternalWritable := 'False'} : Bool;   // Position 20 Roller Transfer Out Reset
      I_Pos20CCSetOutTrf { ExternalAccessible := 'False'; ExternalVisible := 'False'; ExternalWritable := 'False'} : Bool;   // Position 20 Cross Conveyor Transfer Out Set
      I_Pos20CCResOutTrf { ExternalAccessible := 'False'; ExternalVisible := 'False'; ExternalWritable := 'False'} : Bool;   // Position 20 Cross Conveyor Transfer Out Reset
      I_Pos21BodyPresent { ExternalAccessible := 'False'; ExternalVisible := 'False'; ExternalWritable := 'False'} : Bool;   // Position 21 Body Present
      I_Pos21CCResOutTrf { ExternalAccessible := 'False'; ExternalVisible := 'False'; ExternalWritable := 'False'} : Bool;   // Position 21 Cross Conveyor Transfer Out Reset
      I_Pos21RollerSetInTrf { ExternalAccessible := 'False'; ExternalVisible := 'False'; ExternalWritable := 'False'} : Bool;   // Position 21 Roller Transfer In Set
      I_Pos21RollerResInTrf { ExternalAccessible := 'False'; ExternalVisible := 'False'; ExternalWritable := 'False'} : Bool;   // Position 21 Roller Transfer In Reset
      I_Pos21CCResInTrf { ExternalAccessible := 'False'; ExternalVisible := 'False'; ExternalWritable := 'False'} : Bool;   // Position 21 Cross Conveyor Transfer In Reset
      I_Pos21CCSetInTrf { ExternalAccessible := 'False'; ExternalVisible := 'False'; ExternalWritable := 'False'} : Bool;   // Position 21 Cross Conveyor Transfer In Set
      I_Pos21RollerSetOutTrf { ExternalAccessible := 'False'; ExternalVisible := 'False'; ExternalWritable := 'False'} : Bool;   // Position 21 Roller Transfer Out Set
      I_Pos21RollerResOutTrf { ExternalAccessible := 'False'; ExternalVisible := 'False'; ExternalWritable := 'False'} : Bool;   // Position 21 Roller Transfer Out Reset
      I_Pos21CCSetOutTrf { ExternalAccessible := 'False'; ExternalVisible := 'False'; ExternalWritable := 'False'} : Bool;   // Position 21 Cross Conveyor Transfer Out Set
      I_Pos22BodyPresent { ExternalAccessible := 'False'; ExternalVisible := 'False'; ExternalWritable := 'False'} : Bool;   // Position 22 Body Present
      I_Pos22CCResOutTrf { ExternalAccessible := 'False'; ExternalVisible := 'False'; ExternalWritable := 'False'} : Bool;   // Position 22 Cross Conveyor Transfer Out Reset
      I_Pos22RollerSetInTrf { ExternalAccessible := 'False'; ExternalVisible := 'False'; ExternalWritable := 'False'} : Bool;   // Position 22 Roller Transfer In Set
      I_Pos22RollerResInTrf { ExternalAccessible := 'False'; ExternalVisible := 'False'; ExternalWritable := 'False'} : Bool;   // Position 22 Roller Transfer In Reset
      I_Pos22CCResInTrf { ExternalAccessible := 'False'; ExternalVisible := 'False'; ExternalWritable := 'False'} : Bool;   // Position 22 Cross Conveyor Transfer In Reset
      I_Pos22CCSetInTrf { ExternalAccessible := 'False'; ExternalVisible := 'False'; ExternalWritable := 'False'} : Bool;   // Position 22 Cross Conveyor Transfer In Set
      I_Pos22RollerSetOutTrf { ExternalAccessible := 'False'; ExternalVisible := 'False'; ExternalWritable := 'False'} : Bool;   // Position 22 Roller Transfer Out Set
      I_Pos22RollerResOutTrf { ExternalAccessible := 'False'; ExternalVisible := 'False'; ExternalWritable := 'False'} : Bool;   // Position 22 Roller Transfer Out Reset
      I_Pos22CCSetOutTrf { ExternalAccessible := 'False'; ExternalVisible := 'False'; ExternalWritable := 'False'} : Bool;   // Position 22 Cross Conveyor Transfer Out Set
      I_Pos23BodyPresent { ExternalAccessible := 'False'; ExternalVisible := 'False'; ExternalWritable := 'False'} : Bool;   // Position 23 Body Present
      I_Pos23CCResOutTrf { ExternalAccessible := 'False'; ExternalVisible := 'False'; ExternalWritable := 'False'} : Bool;   // Position 23 Cross Conveyor Transfer Out Reset
      I_Pos23RollerSetInTrf { ExternalAccessible := 'False'; ExternalVisible := 'False'; ExternalWritable := 'False'} : Bool;   // Position 23 Roller Transfer In Set
      I_Pos23RollerResInTrf { ExternalAccessible := 'False'; ExternalVisible := 'False'; ExternalWritable := 'False'} : Bool;   // Position 23 Roller Transfer In Reset
      I_Pos23CCResInTrf { ExternalAccessible := 'False'; ExternalVisible := 'False'; ExternalWritable := 'False'} : Bool;   // Position 23 Cross Conveyor Transfer In Reset
      I_Pos23CCSetInTrf { ExternalAccessible := 'False'; ExternalVisible := 'False'; ExternalWritable := 'False'} : Bool;   // Position 23 Cross Conveyor Transfer In Set
      I_Pos23RollerSetOutTrf { ExternalAccessible := 'False'; ExternalVisible := 'False'; ExternalWritable := 'False'} : Bool;   // Position 23 Roller Transfer Out Set
      I_Pos23RollerResOutTrf { ExternalAccessible := 'False'; ExternalVisible := 'False'; ExternalWritable := 'False'} : Bool;   // Position 23 Roller Transfer Out Reset
      I_Pos23CCSetOutTrf { ExternalAccessible := 'False'; ExternalVisible := 'False'; ExternalWritable := 'False'} : Bool;   // Position 23 Cross Conveyor Transfer Out Set
      I_Pos24BodyPresent { ExternalAccessible := 'False'; ExternalVisible := 'False'; ExternalWritable := 'False'} : Bool;   // Position 24 Body Present
      I_Pos24CCResOutTrf { ExternalAccessible := 'False'; ExternalVisible := 'False'; ExternalWritable := 'False'} : Bool;   // Position 24 Cross Conveyor Transfer Out Reset
      I_Pos24RollerSetInTrf { ExternalAccessible := 'False'; ExternalVisible := 'False'; ExternalWritable := 'False'} : Bool;   // Position 24 Roller Transfer In Set
      I_Pos24RollerResInTrf { ExternalAccessible := 'False'; ExternalVisible := 'False'; ExternalWritable := 'False'} : Bool;   // Position 24 Roller Transfer In Reset
      I_Pos24CCResInTrf { ExternalAccessible := 'False'; ExternalVisible := 'False'; ExternalWritable := 'False'} : Bool;   // Position 24 Cross Conveyor Transfer In Reset
      I_Pos24CCSetInTrf { ExternalAccessible := 'False'; ExternalVisible := 'False'; ExternalWritable := 'False'} : Bool;   // Position 24 Cross Conveyor Transfer In Set
      I_Pos24RollerSetOutTrf { ExternalAccessible := 'False'; ExternalVisible := 'False'; ExternalWritable := 'False'} : Bool;   // Position 24 Roller Transfer Out Set
      I_Pos24RollerResOutTrf { ExternalAccessible := 'False'; ExternalVisible := 'False'; ExternalWritable := 'False'} : Bool;   // Position 24 Roller Transfer Out Reset
      I_Pos24CCSetOutTrf { ExternalAccessible := 'False'; ExternalVisible := 'False'; ExternalWritable := 'False'} : Bool;   // Position 24 Cross Conveyor Transfer Out Set
      I_Pos25BodyPresent { ExternalAccessible := 'False'; ExternalVisible := 'False'; ExternalWritable := 'False'} : Bool;   // Position 25 Body Present
      I_Pos25CCResOutTrf { ExternalAccessible := 'False'; ExternalVisible := 'False'; ExternalWritable := 'False'} : Bool;   // Position 25 Cross Conveyor Transfer Out Reset
      I_Pos25RollerSetInTrf { ExternalAccessible := 'False'; ExternalVisible := 'False'; ExternalWritable := 'False'} : Bool;   // Position 25 Roller Transfer In Set
      I_Pos25RollerResInTrf { ExternalAccessible := 'False'; ExternalVisible := 'False'; ExternalWritable := 'False'} : Bool;   // Position 25 Roller Transfer In Reset
      I_Pos25CCResInTrf { ExternalAccessible := 'False'; ExternalVisible := 'False'; ExternalWritable := 'False'} : Bool;   // Position 25 Cross Conveyor Transfer In Reset
      I_Pos25CCSetInTrf { ExternalAccessible := 'False'; ExternalVisible := 'False'; ExternalWritable := 'False'} : Bool;   // Position 25 Cross Conveyor Transfer In Set
      I_Pos25RollerSetOutTrf { ExternalAccessible := 'False'; ExternalVisible := 'False'; ExternalWritable := 'False'} : Bool;   // Position 25 Roller Transfer Out Set
      I_Pos25RollerResOutTrf { ExternalAccessible := 'False'; ExternalVisible := 'False'; ExternalWritable := 'False'} : Bool;   // Position 25 Roller Transfer Out Reset
      I_Pos25CCSetOutTrf { ExternalAccessible := 'False'; ExternalVisible := 'False'; ExternalWritable := 'False'} : Bool;   // Position 25 Cross Conveyor Transfer Out Set
      I_Pos26BodyPresent { ExternalAccessible := 'False'; ExternalVisible := 'False'; ExternalWritable := 'False'} : Bool;   // Position 26 Body Present
      I_Pos26CCResOutTrf { ExternalAccessible := 'False'; ExternalVisible := 'False'; ExternalWritable := 'False'} : Bool;   // Position 26 Cross Conveyor Transfer Out Reset
      I_Pos26RollerSetInTrf { ExternalAccessible := 'False'; ExternalVisible := 'False'; ExternalWritable := 'False'} : Bool;   // Position 26 Roller Transfer In Set
      I_Pos26RollerResInTrf { ExternalAccessible := 'False'; ExternalVisible := 'False'; ExternalWritable := 'False'} : Bool;   // Position 26 Roller Transfer In Reset
      I_Pos26CCResInTrf { ExternalAccessible := 'False'; ExternalVisible := 'False'; ExternalWritable := 'False'} : Bool;   // Position 26 Cross Conveyor Transfer In Reset
      I_Pos26CCSetInTrf { ExternalAccessible := 'False'; ExternalVisible := 'False'; ExternalWritable := 'False'} : Bool;   // Position 26 Cross Conveyor Transfer In Set
      I_Pos26RollerSetOutTrf { ExternalAccessible := 'False'; ExternalVisible := 'False'; ExternalWritable := 'False'} : Bool;   // Position 26 Roller Transfer Out Set
      I_Pos26RollerResOutTrf { ExternalAccessible := 'False'; ExternalVisible := 'False'; ExternalWritable := 'False'} : Bool;   // Position 26 Roller Transfer Out Reset
      I_Pos26CCSetOutTrf { ExternalAccessible := 'False'; ExternalVisible := 'False'; ExternalWritable := 'False'} : Bool;   // Position 26 Cross Conveyor Transfer Out Set
      I_Pos27BodyPresent { ExternalAccessible := 'False'; ExternalVisible := 'False'; ExternalWritable := 'False'} : Bool;   // Position 27 Body Present
      I_Pos27CCResOutTrf { ExternalAccessible := 'False'; ExternalVisible := 'False'; ExternalWritable := 'False'} : Bool;   // Position 27 Cross Conveyor Transfer Out Reset
      I_Pos27RollerSetInTrf { ExternalAccessible := 'False'; ExternalVisible := 'False'; ExternalWritable := 'False'} : Bool;   // Position 27 Roller Transfer In Set
      I_Pos27RollerResInTrf { ExternalAccessible := 'False'; ExternalVisible := 'False'; ExternalWritable := 'False'} : Bool;   // Position 27 Roller Transfer In Reset
      I_Pos27CCResInTrf { ExternalAccessible := 'False'; ExternalVisible := 'False'; ExternalWritable := 'False'} : Bool;   // Position 27 Cross Conveyor Transfer In Reset
      I_Pos27CCSetInTrf { ExternalAccessible := 'False'; ExternalVisible := 'False'; ExternalWritable := 'False'} : Bool;   // Position 27 Cross Conveyor Transfer In Set
      I_Pos27RollerSetOutTrf { ExternalAccessible := 'False'; ExternalVisible := 'False'; ExternalWritable := 'False'} : Bool;   // Position 27 Roller Transfer Out Set
      I_Pos27RollerResOutTrf { ExternalAccessible := 'False'; ExternalVisible := 'False'; ExternalWritable := 'False'} : Bool;   // Position 27 Roller Transfer Out Reset
      I_Pos27CCSetOutTrf { ExternalAccessible := 'False'; ExternalVisible := 'False'; ExternalWritable := 'False'} : Bool;   // Position 27 Cross Conveyor Transfer Out Set
      I_Pos28BodyPresent { ExternalAccessible := 'False'; ExternalVisible := 'False'; ExternalWritable := 'False'} : Bool;   // Position 28 Body Present
      I_Pos28CCResOutTrf { ExternalAccessible := 'False'; ExternalVisible := 'False'; ExternalWritable := 'False'} : Bool;   // Position 28 Cross Conveyor Transfer Out Reset
      I_Pos28RollerSetInTrf { ExternalAccessible := 'False'; ExternalVisible := 'False'; ExternalWritable := 'False'} : Bool;   // Position 28 Roller Transfer In Set
      I_Pos28RollerResInTrf { ExternalAccessible := 'False'; ExternalVisible := 'False'; ExternalWritable := 'False'} : Bool;   // Position 28 Roller Transfer In Reset
      I_Pos28CCResInTrf { ExternalAccessible := 'False'; ExternalVisible := 'False'; ExternalWritable := 'False'} : Bool;   // Position 28 Cross Conveyor Transfer In Reset
      I_Pos28CCSetInTrf { ExternalAccessible := 'False'; ExternalVisible := 'False'; ExternalWritable := 'False'} : Bool;   // Position 28 Cross Conveyor Transfer In Set
      I_Pos28RollerSetOutTrf { ExternalAccessible := 'False'; ExternalVisible := 'False'; ExternalWritable := 'False'} : Bool;   // Position 28 Roller Transfer Out Set
      I_Pos28RollerResOutTrf { ExternalAccessible := 'False'; ExternalVisible := 'False'; ExternalWritable := 'False'} : Bool;   // Position 28 Roller Transfer Out Reset
      I_Pos28CCSetOutTrf { ExternalAccessible := 'False'; ExternalVisible := 'False'; ExternalWritable := 'False'} : Bool;   // Position 28 Cross Conveyor Transfer Out Set
      I_Pos29BodyPresent { ExternalAccessible := 'False'; ExternalVisible := 'False'; ExternalWritable := 'False'} : Bool;   // Position 29 Body Present
      I_Pos29CCResOutTrf { ExternalAccessible := 'False'; ExternalVisible := 'False'; ExternalWritable := 'False'} : Bool;   // Position 29 Cross Conveyor Transfer Out Reset
      I_Pos29RollerSetInTrf { ExternalAccessible := 'False'; ExternalVisible := 'False'; ExternalWritable := 'False'} : Bool;   // Position 29 Roller Transfer In Set
      I_Pos29RollerResInTrf { ExternalAccessible := 'False'; ExternalVisible := 'False'; ExternalWritable := 'False'} : Bool;   // Position 29 Roller Transfer In Reset
      I_Pos29CCResInTrf { ExternalAccessible := 'False'; ExternalVisible := 'False'; ExternalWritable := 'False'} : Bool;   // Position 29 Cross Conveyor Transfer In Reset
      I_Pos29CCSetInTrf { ExternalAccessible := 'False'; ExternalVisible := 'False'; ExternalWritable := 'False'} : Bool;   // Position 29 Cross Conveyor Transfer In Set
      I_Pos29RollerSetOutTrf { ExternalAccessible := 'False'; ExternalVisible := 'False'; ExternalWritable := 'False'} : Bool;   // Position 29 Roller Transfer Out Set
      I_Pos29RollerResOutTrf { ExternalAccessible := 'False'; ExternalVisible := 'False'; ExternalWritable := 'False'} : Bool;   // Position 29 Roller Transfer Out Reset
      I_Pos29CCSetOutTrf { ExternalAccessible := 'False'; ExternalVisible := 'False'; ExternalWritable := 'False'} : Bool;   // Position 29 Cross Conveyor Transfer Out Set
      I_Pos30BodyPresent { ExternalAccessible := 'False'; ExternalVisible := 'False'; ExternalWritable := 'False'} : Bool;   // Position 30 Body Present
      I_Pos30CCResOutTrf { ExternalAccessible := 'False'; ExternalVisible := 'False'; ExternalWritable := 'False'} : Bool;   // Position 30 Cross Conveyor Transfer Out Reset
      I_Pos30RollerSetInTrf { ExternalAccessible := 'False'; ExternalVisible := 'False'; ExternalWritable := 'False'} : Bool;   // Position 30 Roller Transfer In Set
      I_Pos30RollerResInTrf { ExternalAccessible := 'False'; ExternalVisible := 'False'; ExternalWritable := 'False'} : Bool;   // Position 30 Roller Transfer In Reset
      I_Pos30CCResInTrf { ExternalAccessible := 'False'; ExternalVisible := 'False'; ExternalWritable := 'False'} : Bool;   // Position 30 Cross Conveyor Transfer In Reset
      I_Pos30CCSetInTrf { ExternalAccessible := 'False'; ExternalVisible := 'False'; ExternalWritable := 'False'} : Bool;   // Position 30 Cross Conveyor Transfer In Set
      I_Pos30RollerSetOutTrf { ExternalAccessible := 'False'; ExternalVisible := 'False'; ExternalWritable := 'False'} : Bool;   // Position 30 Roller Transfer Out Set
      I_Pos30RollerResOutTrf { ExternalAccessible := 'False'; ExternalVisible := 'False'; ExternalWritable := 'False'} : Bool;   // Position 30 Roller Transfer Out Reset
      I_Pos30CCSetOutTrf { ExternalAccessible := 'False'; ExternalVisible := 'False'; ExternalWritable := 'False'} : Bool;   // Position 30 Cross Conveyor Transfer Out Set
      I_Pos31BodyPresent { ExternalAccessible := 'False'; ExternalVisible := 'False'; ExternalWritable := 'False'} : Bool;   // Position 31 Body Present
      I_Pos31CCResOutTrf { ExternalAccessible := 'False'; ExternalVisible := 'False'; ExternalWritable := 'False'} : Bool;   // Position 31 Cross Conveyor Transfer Out Reset
      I_Pos31RollerSetInTrf { ExternalAccessible := 'False'; ExternalVisible := 'False'; ExternalWritable := 'False'} : Bool;   // Position 31 Roller Transfer In Set
      I_Pos31RollerResInTrf { ExternalAccessible := 'False'; ExternalVisible := 'False'; ExternalWritable := 'False'} : Bool;   // Position 31 Roller Transfer In Reset
      I_Pos31CCResInTrf { ExternalAccessible := 'False'; ExternalVisible := 'False'; ExternalWritable := 'False'} : Bool;   // Position 31 Cross Conveyor Transfer In Reset
      I_Pos31CCSetInTrf { ExternalAccessible := 'False'; ExternalVisible := 'False'; ExternalWritable := 'False'} : Bool;   // Position 31 Cross Conveyor Transfer In Set
      I_Pos31RollerSetOutTrf { ExternalAccessible := 'False'; ExternalVisible := 'False'; ExternalWritable := 'False'} : Bool;   // Position 31 Roller Transfer Out Set
      I_Pos31RollerResOutTrf { ExternalAccessible := 'False'; ExternalVisible := 'False'; ExternalWritable := 'False'} : Bool;   // Position 31 Roller Transfer Out Reset
      I_Pos31CCSetOutTrf { ExternalAccessible := 'False'; ExternalVisible := 'False'; ExternalWritable := 'False'} : Bool;   // Position 31 Cross Conveyor Transfer Out Set
      I_Pos32BodyPresent { ExternalAccessible := 'False'; ExternalVisible := 'False'; ExternalWritable := 'False'} : Bool;   // Position 32 Body Present
      I_Pos32CCResOutTrf { ExternalAccessible := 'False'; ExternalVisible := 'False'; ExternalWritable := 'False'} : Bool;   // Position 32 Cross Conveyor Transfer Out Reset
      I_Pos32RollerSetInTrf { ExternalAccessible := 'False'; ExternalVisible := 'False'; ExternalWritable := 'False'} : Bool;   // Position 32 Roller Transfer In Set
      I_Pos32RollerResInTrf { ExternalAccessible := 'False'; ExternalVisible := 'False'; ExternalWritable := 'False'} : Bool;   // Position 32 Roller Transfer In Reset
      I_Pos32CCResInTrf { ExternalAccessible := 'False'; ExternalVisible := 'False'; ExternalWritable := 'False'} : Bool;   // Position 32 Cross Conveyor Transfer In Reset
      I_Pos32CCSetInTrf { ExternalAccessible := 'False'; ExternalVisible := 'False'; ExternalWritable := 'False'} : Bool;   // Position 32 Cross Conveyor Transfer In Set
      I_Pos32RollerSetOutTrf { ExternalAccessible := 'False'; ExternalVisible := 'False'; ExternalWritable := 'False'} : Bool;   // Position 32 Roller Transfer Out Set
      I_Pos32RollerResOutTrf { ExternalAccessible := 'False'; ExternalVisible := 'False'; ExternalWritable := 'False'} : Bool;   // Position 32 Roller Transfer Out Reset
      I_Pos32CCSetOutTrf { ExternalAccessible := 'False'; ExternalVisible := 'False'; ExternalWritable := 'False'} : Bool;   // Position 32 Cross Conveyor Transfer Out Set
      I_Pos33BodyPresent { ExternalAccessible := 'False'; ExternalVisible := 'False'; ExternalWritable := 'False'} : Bool;   // Position 33 Body Present
      I_Pos33CCResOutTrf { ExternalAccessible := 'False'; ExternalVisible := 'False'; ExternalWritable := 'False'} : Bool;   // Position 33 Cross Conveyor Transfer Out Reset
      I_Pos33RollerSetInTrf { ExternalAccessible := 'False'; ExternalVisible := 'False'; ExternalWritable := 'False'} : Bool;   // Position 33 Roller Transfer In Set
      I_Pos33RollerResInTrf { ExternalAccessible := 'False'; ExternalVisible := 'False'; ExternalWritable := 'False'} : Bool;   // Position 33 Roller Transfer In Reset
      I_Pos33CCResInTrf { ExternalAccessible := 'False'; ExternalVisible := 'False'; ExternalWritable := 'False'} : Bool;   // Position 33 Cross Conveyor Transfer In Reset
      I_Pos33CCSetInTrf { ExternalAccessible := 'False'; ExternalVisible := 'False'; ExternalWritable := 'False'} : Bool;   // Position 33 Cross Conveyor Transfer In Set
      I_Pos33RollerSetOutTrf { ExternalAccessible := 'False'; ExternalVisible := 'False'; ExternalWritable := 'False'} : Bool;   // Position 33 Roller Transfer Out Set
      I_Pos33RollerResOutTrf { ExternalAccessible := 'False'; ExternalVisible := 'False'; ExternalWritable := 'False'} : Bool;   // Position 33 Roller Transfer Out Reset
      I_Pos33CCSetOutTrf { ExternalAccessible := 'False'; ExternalVisible := 'False'; ExternalWritable := 'False'} : Bool;   // Position 33 Cross Conveyor Transfer Out Set
      I_Pos34BodyPresent { ExternalAccessible := 'False'; ExternalVisible := 'False'; ExternalWritable := 'False'} : Bool;   // Position 34 Body Present
      I_Pos34CCResOutTrf { ExternalAccessible := 'False'; ExternalVisible := 'False'; ExternalWritable := 'False'} : Bool;   // Position 34 Cross Conveyor Transfer Out Reset
      I_Pos34RollerSetInTrf { ExternalAccessible := 'False'; ExternalVisible := 'False'; ExternalWritable := 'False'} : Bool;   // Position 34 Roller Transfer In Set
      I_Pos34RollerResInTrf { ExternalAccessible := 'False'; ExternalVisible := 'False'; ExternalWritable := 'False'} : Bool;   // Position 34 Roller Transfer In Reset
      I_Pos34CCResInTrf { ExternalAccessible := 'False'; ExternalVisible := 'False'; ExternalWritable := 'False'} : Bool;   // Position 34 Cross Conveyor Transfer In Reset
      I_Pos34CCSetInTrf { ExternalAccessible := 'False'; ExternalVisible := 'False'; ExternalWritable := 'False'} : Bool;   // Position 34 Cross Conveyor Transfer In Set
      I_Pos34RollerSetOutTrf { ExternalAccessible := 'False'; ExternalVisible := 'False'; ExternalWritable := 'False'} : Bool;   // Position 34 Roller Transfer Out Set
      I_Pos34RollerResOutTrf { ExternalAccessible := 'False'; ExternalVisible := 'False'; ExternalWritable := 'False'} : Bool;   // Position 34 Roller Transfer Out Reset
      I_Pos34CCSetOutTrf { ExternalAccessible := 'False'; ExternalVisible := 'False'; ExternalWritable := 'False'} : Bool;   // Position 34 Cross Conveyor Transfer Out Set
      I_Pos35BodyPresent { ExternalAccessible := 'False'; ExternalVisible := 'False'; ExternalWritable := 'False'} : Bool;   // Position 35 Body Present
      I_Pos35CCResOutTrf { ExternalAccessible := 'False'; ExternalVisible := 'False'; ExternalWritable := 'False'} : Bool;   // Position 35 Cross Conveyor Transfer Out Reset
      I_Pos35RollerSetInTrf { ExternalAccessible := 'False'; ExternalVisible := 'False'; ExternalWritable := 'False'} : Bool;   // Position 35 Roller Transfer In Set
      I_Pos35RollerResInTrf { ExternalAccessible := 'False'; ExternalVisible := 'False'; ExternalWritable := 'False'} : Bool;   // Position 35 Roller Transfer In Reset
      I_Pos35CCResInTrf { ExternalAccessible := 'False'; ExternalVisible := 'False'; ExternalWritable := 'False'} : Bool;   // Position 35 Cross Conveyor Transfer In Reset
      I_Pos35CCSetInTrf { ExternalAccessible := 'False'; ExternalVisible := 'False'; ExternalWritable := 'False'} : Bool;   // Position 35 Cross Conveyor Transfer In Set
      I_Pos35RollerSetOutTrf { ExternalAccessible := 'False'; ExternalVisible := 'False'; ExternalWritable := 'False'} : Bool;   // Position 35 Roller Transfer Out Set
      I_Pos35RollerResOutTrf { ExternalAccessible := 'False'; ExternalVisible := 'False'; ExternalWritable := 'False'} : Bool;   // Position 35 Roller Transfer Out Reset
      I_Pos35CCSetOutTrf { ExternalAccessible := 'False'; ExternalVisible := 'False'; ExternalWritable := 'False'} : Bool;   // Position 35 Cross Conveyor Transfer Out Set
      I_Pos36BodyPresent { ExternalAccessible := 'False'; ExternalVisible := 'False'; ExternalWritable := 'False'} : Bool;   // Position 36 Body Present
      I_Pos36CCResOutTrf { ExternalAccessible := 'False'; ExternalVisible := 'False'; ExternalWritable := 'False'} : Bool;   // Position 36 Cross Conveyor Transfer Out Reset
      I_Pos36RollerSetInTrf { ExternalAccessible := 'False'; ExternalVisible := 'False'; ExternalWritable := 'False'} : Bool;   // Position 36 Roller Transfer In Set
      I_Pos36RollerResInTrf { ExternalAccessible := 'False'; ExternalVisible := 'False'; ExternalWritable := 'False'} : Bool;   // Position 36 Roller Transfer In Reset
      I_Pos36CCResInTrf { ExternalAccessible := 'False'; ExternalVisible := 'False'; ExternalWritable := 'False'} : Bool;   // Position 36 Cross Conveyor Transfer In Reset
      I_Pos36CCSetInTrf { ExternalAccessible := 'False'; ExternalVisible := 'False'; ExternalWritable := 'False'} : Bool;   // Position 36 Cross Conveyor Transfer In Set
      I_Pos36RollerSetOutTrf { ExternalAccessible := 'False'; ExternalVisible := 'False'; ExternalWritable := 'False'} : Bool;   // Position 36 Roller Transfer Out Set
      I_Pos36RollerResOutTrf { ExternalAccessible := 'False'; ExternalVisible := 'False'; ExternalWritable := 'False'} : Bool;   // Position 36 Roller Transfer Out Reset
      I_Pos36CCSetOutTrf { ExternalAccessible := 'False'; ExternalVisible := 'False'; ExternalWritable := 'False'} : Bool;   // Position 36 Cross Conveyor Transfer Out Set
      I_Pos37BodyPresent { ExternalAccessible := 'False'; ExternalVisible := 'False'; ExternalWritable := 'False'} : Bool;   // Position 37 Body Present
      I_Pos37CCResOutTrf { ExternalAccessible := 'False'; ExternalVisible := 'False'; ExternalWritable := 'False'} : Bool;   // Position 37 Cross Conveyor Transfer Out Reset
      I_Pos37RollerSetInTrf { ExternalAccessible := 'False'; ExternalVisible := 'False'; ExternalWritable := 'False'} : Bool;   // Position 37 Roller Transfer In Set
      I_Pos37RollerResInTrf { ExternalAccessible := 'False'; ExternalVisible := 'False'; ExternalWritable := 'False'} : Bool;   // Position 37 Roller Transfer In Reset
      I_Pos37CCResInTrf { ExternalAccessible := 'False'; ExternalVisible := 'False'; ExternalWritable := 'False'} : Bool;   // Position 37 Cross Conveyor Transfer In Reset
      I_Pos37CCSetInTrf { ExternalAccessible := 'False'; ExternalVisible := 'False'; ExternalWritable := 'False'} : Bool;   // Position 37 Cross Conveyor Transfer In Set
      I_Pos37RollerSetOutTrf { ExternalAccessible := 'False'; ExternalVisible := 'False'; ExternalWritable := 'False'} : Bool;   // Position 37 Roller Transfer Out Set
      I_Pos37RollerResOutTrf { ExternalAccessible := 'False'; ExternalVisible := 'False'; ExternalWritable := 'False'} : Bool;   // Position 37 Roller Transfer Out Reset
      I_Pos37CCSetOutTrf { ExternalAccessible := 'False'; ExternalVisible := 'False'; ExternalWritable := 'False'} : Bool;   // Position 37 Cross Conveyor Transfer Out Set
      I_Pos38BodyPresent { ExternalAccessible := 'False'; ExternalVisible := 'False'; ExternalWritable := 'False'} : Bool;   // Position 38 Body Present
      I_Pos38CCResOutTrf { ExternalAccessible := 'False'; ExternalVisible := 'False'; ExternalWritable := 'False'} : Bool;   // Position 38 Cross Conveyor Transfer Out Reset
      I_Pos38RollerSetInTrf { ExternalAccessible := 'False'; ExternalVisible := 'False'; ExternalWritable := 'False'} : Bool;   // Position 38 Roller Transfer In Set
      I_Pos38RollerResInTrf { ExternalAccessible := 'False'; ExternalVisible := 'False'; ExternalWritable := 'False'} : Bool;   // Position 38 Roller Transfer In Reset
      I_Pos38CCResInTrf { ExternalAccessible := 'False'; ExternalVisible := 'False'; ExternalWritable := 'False'} : Bool;   // Position 38 Cross Conveyor Transfer In Reset
      I_Pos38CCSetInTrf { ExternalAccessible := 'False'; ExternalVisible := 'False'; ExternalWritable := 'False'} : Bool;   // Position 38 Cross Conveyor Transfer In Set
      I_Pos38RollerSetOutTrf { ExternalAccessible := 'False'; ExternalVisible := 'False'; ExternalWritable := 'False'} : Bool;   // Position 38 Roller Transfer Out Set
      I_Pos38RollerResOutTrf { ExternalAccessible := 'False'; ExternalVisible := 'False'; ExternalWritable := 'False'} : Bool;   // Position 38 Roller Transfer Out Reset
      I_Pos38CCSetOutTrf { ExternalAccessible := 'False'; ExternalVisible := 'False'; ExternalWritable := 'False'} : Bool;   // Position 38 Cross Conveyor Transfer Out Set
      I_Pos39BodyPresent { ExternalAccessible := 'False'; ExternalVisible := 'False'; ExternalWritable := 'False'} : Bool;   // Position 39 Body Present
      I_Pos39CCResOutTrf { ExternalAccessible := 'False'; ExternalVisible := 'False'; ExternalWritable := 'False'} : Bool;   // Position 39 Cross Conveyor Transfer Out Reset
      I_Pos39RollerSetInTrf { ExternalAccessible := 'False'; ExternalVisible := 'False'; ExternalWritable := 'False'} : Bool;   // Position 39 Roller Transfer In Set
      I_Pos39RollerResInTrf { ExternalAccessible := 'False'; ExternalVisible := 'False'; ExternalWritable := 'False'} : Bool;   // Position 39 Roller Transfer In Reset
      I_Pos39CCResInTrf { ExternalAccessible := 'False'; ExternalVisible := 'False'; ExternalWritable := 'False'} : Bool;   // Position 39 Cross Conveyor Transfer In Reset
      I_Pos39CCSetInTrf { ExternalAccessible := 'False'; ExternalVisible := 'False'; ExternalWritable := 'False'} : Bool;   // Position 39 Cross Conveyor Transfer In Set
      I_Pos39RollerSetOutTrf { ExternalAccessible := 'False'; ExternalVisible := 'False'; ExternalWritable := 'False'} : Bool;   // Position 39 Roller Transfer Out Set
      I_Pos39RollerResOutTrf { ExternalAccessible := 'False'; ExternalVisible := 'False'; ExternalWritable := 'False'} : Bool;   // Position 39 Roller Transfer Out Reset
      I_Pos39CCSetOutTrf { ExternalAccessible := 'False'; ExternalVisible := 'False'; ExternalWritable := 'False'} : Bool;   // Position 39 Cross Conveyor Transfer Out Set
      I_Pos40BodyPresent { ExternalAccessible := 'False'; ExternalVisible := 'False'; ExternalWritable := 'False'} : Bool;   // Position 40 Body Present
      I_Pos40CCResOutTrf { ExternalAccessible := 'False'; ExternalVisible := 'False'; ExternalWritable := 'False'} : Bool;   // Position 40 Cross Conveyor Transfer Out Reset
      I_Pos40RollerSetInTrf { ExternalAccessible := 'False'; ExternalVisible := 'False'; ExternalWritable := 'False'} : Bool;   // Position 40 Roller Transfer In Set
      I_Pos40RollerResInTrf { ExternalAccessible := 'False'; ExternalVisible := 'False'; ExternalWritable := 'False'} : Bool;   // Position 40 Roller Transfer In Reset
      I_Pos40CCResInTrf { ExternalAccessible := 'False'; ExternalVisible := 'False'; ExternalWritable := 'False'} : Bool;   // Position 40 Cross Conveyor Transfer In Reset
      I_Pos40CCSetInTrf { ExternalAccessible := 'False'; ExternalVisible := 'False'; ExternalWritable := 'False'} : Bool;   // Position 40 Cross Conveyor Transfer In Set
      I_Pos40RollerSetOutTrf { ExternalAccessible := 'False'; ExternalVisible := 'False'; ExternalWritable := 'False'} : Bool;   // Position 40 Roller Transfer Out Set
      I_Pos40RollerResOutTrf { ExternalAccessible := 'False'; ExternalVisible := 'False'; ExternalWritable := 'False'} : Bool;   // Position 40 Roller Transfer Out Reset
      I_Pos40CCSetOutTrf { ExternalAccessible := 'False'; ExternalVisible := 'False'; ExternalWritable := 'False'} : Bool;   // Position 40 Cross Conveyor Transfer Out Set
   END_VAR
   VAR_OUTPUT
      O_CounterValue { ExternalAccessible := 'False'; ExternalVisible := 'False'; ExternalWritable := 'False'} : DInt;   // Counter Value
      O_CounterValueConv1 { ExternalAccessible := 'False'; ExternalVisible := 'False'; ExternalWritable := 'False'} : DInt;   // Counter Value Conveyor 1
      O_CounterValueConv2 { ExternalAccessible := 'False'; ExternalVisible := 'False'; ExternalWritable := 'False'} : DInt;   // Counter Value Conveyor 2
      O_StationFull { ExternalAccessible := 'False'; ExternalVisible := 'False'; ExternalWritable := 'False'} : Bool;   // Zone Full
      O_DynamicMaxActive { ExternalAccessible := 'False'; ExternalVisible := 'False'; ExternalWritable := 'False'} : Bool;   // Dynamic Buffer Active
      O_CounterConv1Alarm { ExternalAccessible := 'False'; ExternalVisible := 'False'; ExternalWritable := 'False'} : Bool;   // Counter Conveyor 1 Value Fault
      O_CounterConv2Alarm { ExternalAccessible := 'False'; ExternalVisible := 'False'; ExternalWritable := 'False'} : Bool;   // Counter Conveyor 2 Value Fault
      O_MaxBody { ExternalAccessible := 'False'; ExternalVisible := 'False'; ExternalWritable := 'False'} : DInt;   // Max Amount of Bodies in the Zone
   END_VAR
   VAR_IN_OUT
      IO_Modes : "Modes";
      H_HMI : "H_HMI";
      H_BodyCounterDynamic : "H_GBBodyCounter";
   END_VAR
   VAR RETAIN
      _CounterConv1 { ExternalAccessible := 'False'; ExternalVisible := 'False'; ExternalWritable := 'False'; S7_SetPoint := 'True'} : CTU_DINT;
      _CounterConv2 { ExternalAccessible := 'False'; ExternalVisible := 'False'; ExternalWritable := 'False'; S7_SetPoint := 'True'} : CTU_DINT;
   END_VAR
   VAR
      Edge { ExternalAccessible := 'False'; ExternalVisible := 'False'; ExternalWritable := 'False'} : Array[0..7] of Bool;   // HM for Edge
      CounterConv1 { ExternalAccessible := 'False'; ExternalVisible := 'False'; ExternalWritable := 'False'} : DInt;   // Counter Conveyor 1
      CounterConv1BelowZero { ExternalAccessible := 'False'; ExternalVisible := 'False'; ExternalWritable := 'False'} : Bool;   // Counter Conveyor 1 Below Zero
      CounterConv1AboveMax { ExternalAccessible := 'False'; ExternalVisible := 'False'; ExternalWritable := 'False'} : Bool;   // Counter Conveyor 1 Above Max
      CounterConv1Add { ExternalAccessible := 'False'; ExternalVisible := 'False'; ExternalWritable := 'False'} : Bool;   // Counter Conveyor 1 Add HMI Button
      CounterConv1Sub { ExternalAccessible := 'False'; ExternalVisible := 'False'; ExternalWritable := 'False'} : Bool;   // Counter Conveyor 1 Subtract HMI Button
      CounterConv1Fault { ExternalAccessible := 'False'; ExternalVisible := 'False'; ExternalWritable := 'False'} : Bool;   // Counter Conveyor 1 Fault
      CounterConv2 { ExternalAccessible := 'False'; ExternalVisible := 'False'; ExternalWritable := 'False'} : DInt;   // Counter Conveyor 2
      CounterConv2BelowZero { ExternalAccessible := 'False'; ExternalVisible := 'False'; ExternalWritable := 'False'} : Bool;   // Counter Conveyor 2 Below Zero
      CounterConv2AboveMax { ExternalAccessible := 'False'; ExternalVisible := 'False'; ExternalWritable := 'False'} : Bool;   // Counter Conveyor 2 Above Max
      CounterConv2Add { ExternalAccessible := 'False'; ExternalVisible := 'False'; ExternalWritable := 'False'} : Bool;   // Counter Conveyor 2 Add HMI Button
      CounterConv2Sub { ExternalAccessible := 'False'; ExternalVisible := 'False'; ExternalWritable := 'False'} : Bool;   // Counter Conveyor 2 Subtract HMI Button
      CounterConv2Fault { ExternalAccessible := 'False'; ExternalVisible := 'False'; ExternalWritable := 'False'} : Bool;   // Counter Conveyor 2 Fault
   END_VAR
   VAR RETAIN
      CounterPos1 { ExternalAccessible := 'False'; ExternalVisible := 'False'; ExternalWritable := 'False'; S7_SetPoint := 'True'} : DInt;
      CounterPos2 { ExternalAccessible := 'False'; ExternalVisible := 'False'; ExternalWritable := 'False'; S7_SetPoint := 'True'} : DInt;
      CounterPos3 { ExternalAccessible := 'False'; ExternalVisible := 'False'; ExternalWritable := 'False'; S7_SetPoint := 'True'} : DInt;
      CounterPos4 { ExternalAccessible := 'False'; ExternalVisible := 'False'; ExternalWritable := 'False'; S7_SetPoint := 'True'} : DInt;
      CounterPos5 { ExternalAccessible := 'False'; ExternalVisible := 'False'; ExternalWritable := 'False'; S7_SetPoint := 'True'} : DInt;
      CounterPos6 { ExternalAccessible := 'False'; ExternalVisible := 'False'; ExternalWritable := 'False'; S7_SetPoint := 'True'} : DInt;
      CounterPos7 { ExternalAccessible := 'False'; ExternalVisible := 'False'; ExternalWritable := 'False'; S7_SetPoint := 'True'} : DInt;
      CounterPos8 { ExternalAccessible := 'False'; ExternalVisible := 'False'; ExternalWritable := 'False'; S7_SetPoint := 'True'} : DInt;
      CounterPos9 { ExternalAccessible := 'False'; ExternalVisible := 'False'; ExternalWritable := 'False'; S7_SetPoint := 'True'} : DInt;
      CounterPos10 { ExternalAccessible := 'False'; ExternalVisible := 'False'; ExternalWritable := 'False'; S7_SetPoint := 'True'} : DInt;
      CounterPos11 { ExternalAccessible := 'False'; ExternalVisible := 'False'; ExternalWritable := 'False'; S7_SetPoint := 'True'} : DInt := 0;
      CounterPos12 { ExternalAccessible := 'False'; ExternalVisible := 'False'; ExternalWritable := 'False'; S7_SetPoint := 'True'} : DInt := 0;
      CounterPos13 { ExternalAccessible := 'False'; ExternalVisible := 'False'; ExternalWritable := 'False'; S7_SetPoint := 'True'} : DInt := 0;
      CounterPos14 { ExternalAccessible := 'False'; ExternalVisible := 'False'; ExternalWritable := 'False'; S7_SetPoint := 'True'} : DInt := 0;
      CounterPos15 { ExternalAccessible := 'False'; ExternalVisible := 'False'; ExternalWritable := 'False'; S7_SetPoint := 'True'} : DInt := 0;
      CounterPos16 { ExternalAccessible := 'False'; ExternalVisible := 'False'; ExternalWritable := 'False'; S7_SetPoint := 'True'} : DInt := 0;
      CounterPos17 { ExternalAccessible := 'False'; ExternalVisible := 'False'; ExternalWritable := 'False'; S7_SetPoint := 'True'} : DInt := 0;
      CounterPos18 { ExternalAccessible := 'False'; ExternalVisible := 'False'; ExternalWritable := 'False'; S7_SetPoint := 'True'} : DInt := 0;
      CounterPos19 { ExternalAccessible := 'False'; ExternalVisible := 'False'; ExternalWritable := 'False'; S7_SetPoint := 'True'} : DInt := 0;
      CounterPos20 { ExternalAccessible := 'False'; ExternalVisible := 'False'; ExternalWritable := 'False'; S7_SetPoint := 'True'} : DInt := 0;
      CounterPos21 { ExternalAccessible := 'False'; ExternalVisible := 'False'; ExternalWritable := 'False'; S7_SetPoint := 'True'} : DInt := 0;
      CounterPos22 { ExternalAccessible := 'False'; ExternalVisible := 'False'; ExternalWritable := 'False'; S7_SetPoint := 'True'} : DInt := 0;
      CounterPos23 { ExternalAccessible := 'False'; ExternalVisible := 'False'; ExternalWritable := 'False'; S7_SetPoint := 'True'} : DInt := 0;
      CounterPos24 { ExternalAccessible := 'False'; ExternalVisible := 'False'; ExternalWritable := 'False'; S7_SetPoint := 'True'} : DInt := 0;
      CounterPos25 { ExternalAccessible := 'False'; ExternalVisible := 'False'; ExternalWritable := 'False'; S7_SetPoint := 'True'} : DInt := 0;
      CounterPos26 { ExternalAccessible := 'False'; ExternalVisible := 'False'; ExternalWritable := 'False'; S7_SetPoint := 'True'} : DInt := 0;
      CounterPos27 { ExternalAccessible := 'False'; ExternalVisible := 'False'; ExternalWritable := 'False'; S7_SetPoint := 'True'} : DInt := 0;
      CounterPos28 { ExternalAccessible := 'False'; ExternalVisible := 'False'; ExternalWritable := 'False'; S7_SetPoint := 'True'} : DInt := 0;
      CounterPos29 { ExternalAccessible := 'False'; ExternalVisible := 'False'; ExternalWritable := 'False'; S7_SetPoint := 'True'} : DInt := 0;
      CounterPos30 { ExternalAccessible := 'False'; ExternalVisible := 'False'; ExternalWritable := 'False'; S7_SetPoint := 'True'} : DInt := 0;
      CounterPos31 { ExternalAccessible := 'False'; ExternalVisible := 'False'; ExternalWritable := 'False'; S7_SetPoint := 'True'} : DInt := 0;
      CounterPos32 { ExternalAccessible := 'False'; ExternalVisible := 'False'; ExternalWritable := 'False'; S7_SetPoint := 'True'} : DInt := 0;
      CounterPos33 { ExternalAccessible := 'False'; ExternalVisible := 'False'; ExternalWritable := 'False'; S7_SetPoint := 'True'} : DInt := 0;
      CounterPos34 { ExternalAccessible := 'False'; ExternalVisible := 'False'; ExternalWritable := 'False'; S7_SetPoint := 'True'} : DInt := 0;
      CounterPos35 { ExternalAccessible := 'False'; ExternalVisible := 'False'; ExternalWritable := 'False'; S7_SetPoint := 'True'} : DInt := 0;
      CounterPos36 { ExternalAccessible := 'False'; ExternalVisible := 'False'; ExternalWritable := 'False'; S7_SetPoint := 'True'} : DInt := 0;
      CounterPos37 { ExternalAccessible := 'False'; ExternalVisible := 'False'; ExternalWritable := 'False'; S7_SetPoint := 'True'} : DInt := 0;
      CounterPos38 { ExternalAccessible := 'False'; ExternalVisible := 'False'; ExternalWritable := 'False'; S7_SetPoint := 'True'} : DInt := 0;
      CounterPos39 { ExternalAccessible := 'False'; ExternalVisible := 'False'; ExternalWritable := 'False'; S7_SetPoint := 'True'} : DInt := 0;
      CounterPos40 { ExternalAccessible := 'False'; ExternalVisible := 'False'; ExternalWritable := 'False'; S7_SetPoint := 'True'} : DInt := 0;
   END_VAR
   VAR
      DirectCounterValue { ExternalAccessible := 'False'; ExternalVisible := 'False'; ExternalWritable := 'False'} : DInt;
      CounterValue { ExternalAccessible := 'False'; ExternalVisible := 'False'; ExternalWritable := 'False'} : DInt;
      _TimerFilterCounterValue { ExternalAccessible := 'False'; ExternalVisible := 'False'; ExternalWritable := 'False'; S7_SetPoint := 'True'} : TON_TIME;
      MaxDynamicDelayTimerUpdate { ExternalAccessible := 'False'; ExternalVisible := 'False'; ExternalWritable := 'False'} : Bool;
      _TimerFilterMaxDynamicTimerValue { ExternalAccessible := 'False'; ExternalVisible := 'False'; ExternalWritable := 'False'; S7_SetPoint := 'True'} : TON_TIME;
      MaxDynamicBody { ExternalAccessible := 'False'; ExternalVisible := 'False'; ExternalWritable := 'False'} : DInt;   // Max Amount of Bodies to Activate Dynamic Buffer
      MaxDynamicDelayTImer { ExternalAccessible := 'False'; ExternalVisible := 'False'; ExternalWritable := 'False'; S7_SetPoint := 'True'} : TON_TIME;
      MaxDynamicDelayTime { ExternalAccessible := 'False'; ExternalVisible := 'False'; ExternalWritable := 'False'; S7_SetPoint := 'True'} : DInt;
      MaxDynamicDelayTimeMem { ExternalAccessible := 'False'; ExternalVisible := 'False'; ExternalWritable := 'False'} : DInt;
      MaxDynamicDelayTimeMs { ExternalAccessible := 'False'; ExternalVisible := 'False'; ExternalWritable := 'False'} : Time;
      DynamicMaxActive { ExternalAccessible := 'False'; ExternalVisible := 'False'; ExternalWritable := 'False'} : Bool;
   END_VAR
   VAR_TEMP   // added for the SCL form of the ladder/FBD networks
      _w1 : Bool;
   END_VAR
BEGIN

REGION Network 1: **** 1 - Inputs **** Inputs from HMI
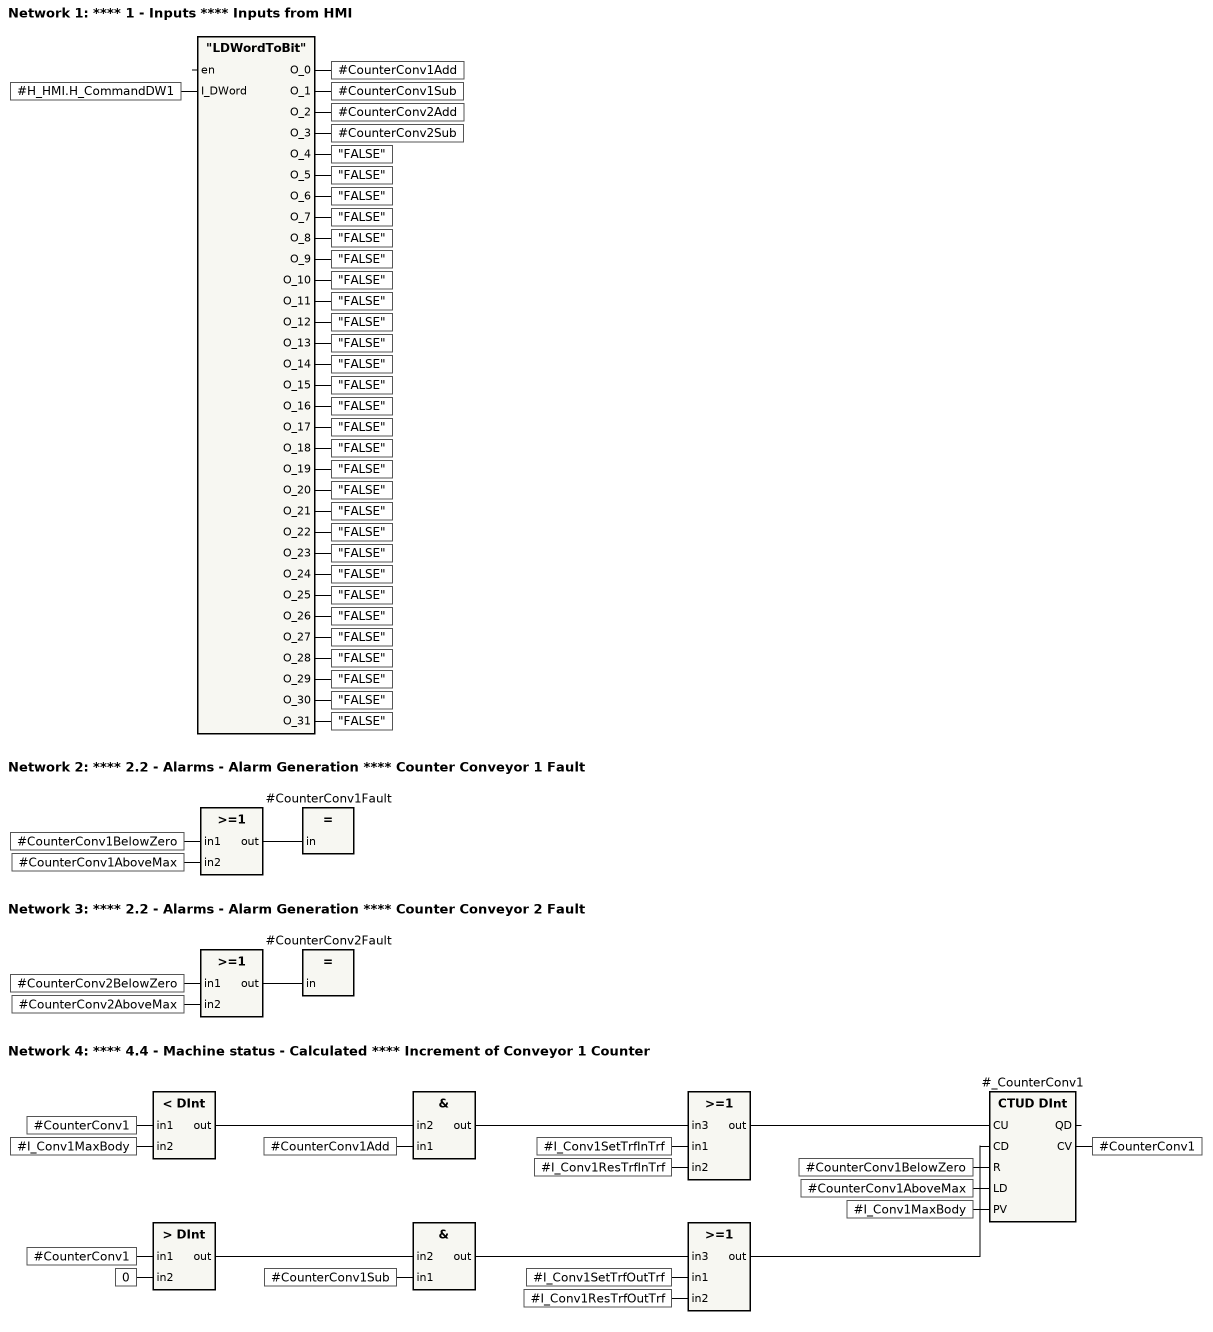
   "LDWordToBit"(I_DWord := #H_HMI.H_CommandDW1,
                 O_0 => #CounterConv1Add,
                 O_1 => #CounterConv1Sub,
                 O_2 => #CounterConv2Add,
                 O_3 => #CounterConv2Sub,
                 O_4 => "FALSE",
                 O_5 => "FALSE",
                 O_6 => "FALSE",
                 O_7 => "FALSE",
                 O_8 => "FALSE",
                 O_9 => "FALSE",
                 O_10 => "FALSE",
                 O_11 => "FALSE",
                 O_12 => "FALSE",
                 O_13 => "FALSE",
                 O_14 => "FALSE",
                 O_15 => "FALSE",
                 O_16 => "FALSE",
                 O_17 => "FALSE",
                 O_18 => "FALSE",
                 O_19 => "FALSE",
                 O_20 => "FALSE",
                 O_21 => "FALSE",
                 O_22 => "FALSE",
                 O_23 => "FALSE",
                 O_24 => "FALSE",
                 O_25 => "FALSE",
                 O_26 => "FALSE",
                 O_27 => "FALSE",
                 O_28 => "FALSE",
                 O_29 => "FALSE",
                 O_30 => "FALSE",
                 O_31 => "FALSE");
END_REGION

REGION Network 2: **** 2.2 - Alarms - Alarm Generation **** Counter Conveyor 1 Fault
   #CounterConv1Fault := #CounterConv1BelowZero OR #CounterConv1AboveMax;
END_REGION

REGION Network 3: **** 2.2 - Alarms - Alarm Generation **** Counter Conveyor 2 Fault
   #CounterConv2Fault := #CounterConv2BelowZero OR #CounterConv2AboveMax;
END_REGION

REGION Network 4: **** 4.4 - Machine status - Calculated **** Increment of Conveyor 1 Counter
   #_CounterConv1(CU := ((#CounterConv1 < #I_Conv1MaxBody) AND #CounterConv1Add) OR #I_Conv1SetTrfInTrf OR #I_Conv1ResTrfInTrf,   // CTUD
                  CD := ((#CounterConv1 > 0) AND #CounterConv1Sub) OR #I_Conv1SetTrfOutTrf OR #I_Conv1ResTrfOutTrf,
                  R := #CounterConv1BelowZero,
                  LD := #CounterConv1AboveMax,
                  PV := #I_Conv1MaxBody,
                  CV => #CounterConv1);
END_REGION

REGION Network 5: **** 4.4 - Machine status - Calculated **** Increment of Conveyor 2 Counter
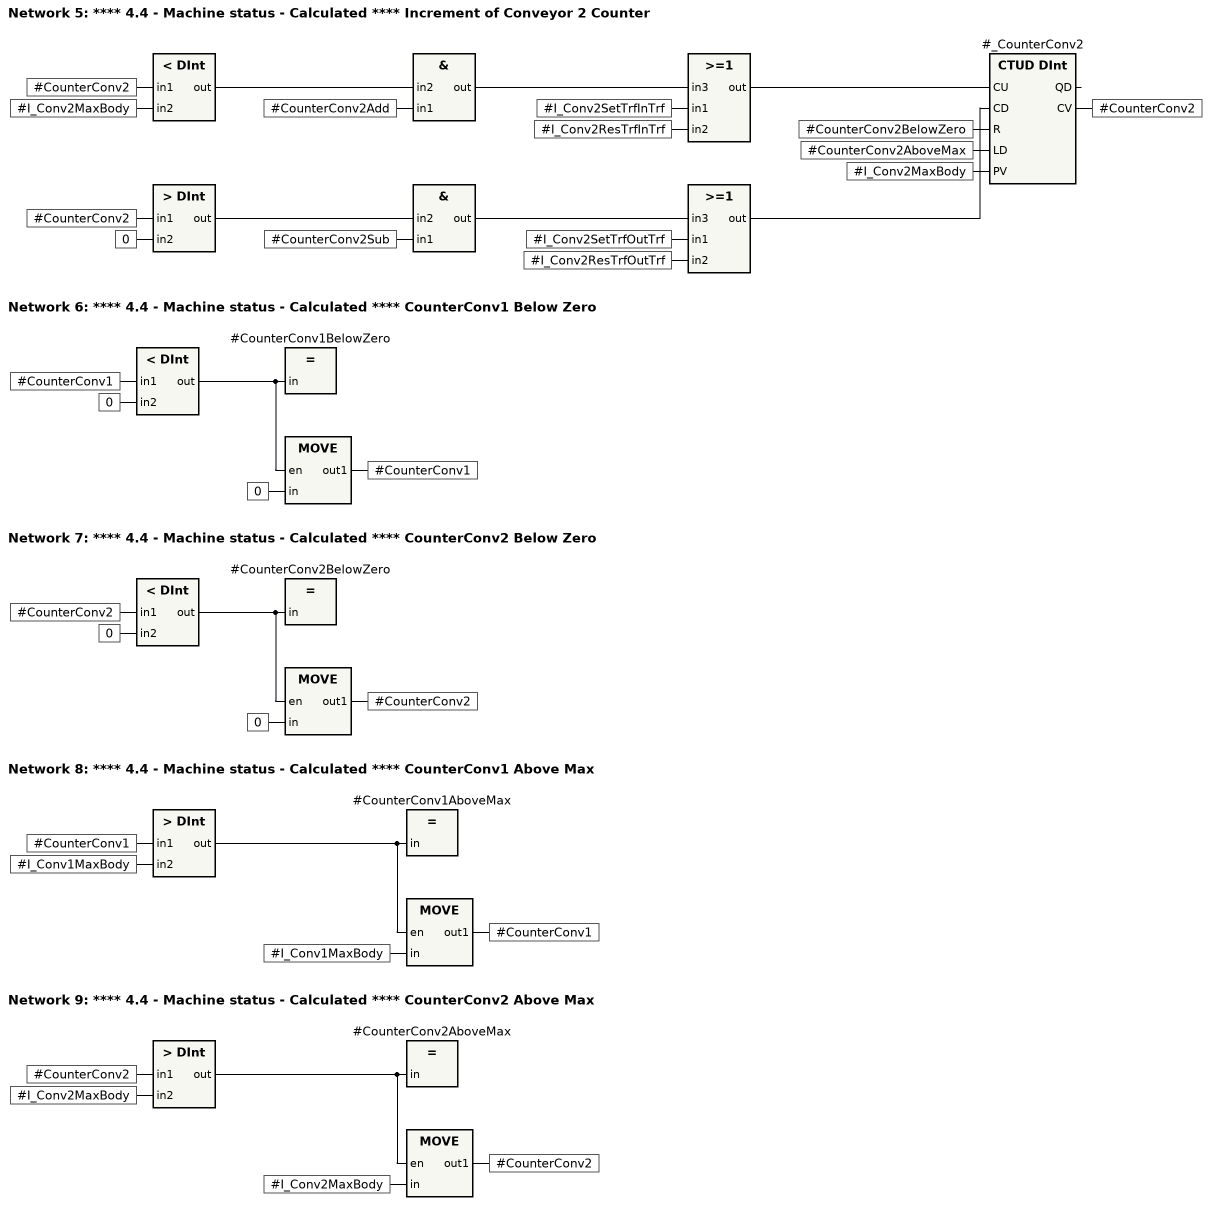
   #_CounterConv2(CU := ((#CounterConv2 < #I_Conv2MaxBody) AND #CounterConv2Add) OR #I_Conv2SetTrfInTrf OR #I_Conv2ResTrfInTrf,   // CTUD
                  CD := ((#CounterConv2 > 0) AND #CounterConv2Sub) OR #I_Conv2SetTrfOutTrf OR #I_Conv2ResTrfOutTrf,
                  R := #CounterConv2BelowZero,
                  LD := #CounterConv2AboveMax,
                  PV := #I_Conv2MaxBody,
                  CV => #CounterConv2);
END_REGION

REGION Network 6: **** 4.4 - Machine status - Calculated **** CounterConv1 Below Zero
   #CounterConv1BelowZero := #CounterConv1 < 0;
   IF #CounterConv1BelowZero THEN #CounterConv1 := 0; END_IF;
END_REGION

REGION Network 7: **** 4.4 - Machine status - Calculated **** CounterConv2 Below Zero
   #CounterConv2BelowZero := #CounterConv2 < 0;
   IF #CounterConv2BelowZero THEN #CounterConv2 := 0; END_IF;
END_REGION

REGION Network 8: **** 4.4 - Machine status - Calculated **** CounterConv1 Above Max
   #CounterConv1AboveMax := #CounterConv1 > #I_Conv1MaxBody;
   IF #CounterConv1AboveMax THEN #CounterConv1 := #I_Conv1MaxBody; END_IF;
END_REGION

REGION Network 9: **** 4.4 - Machine status - Calculated **** CounterConv2 Above Max
   #CounterConv2AboveMax := #CounterConv2 > #I_Conv2MaxBody;
   IF #CounterConv2AboveMax THEN #CounterConv2 := #I_Conv2MaxBody; END_IF;
END_REGION

REGION Network 10: **** 4.4 - Machine status - Calculated **** Counters Equipment to Zero
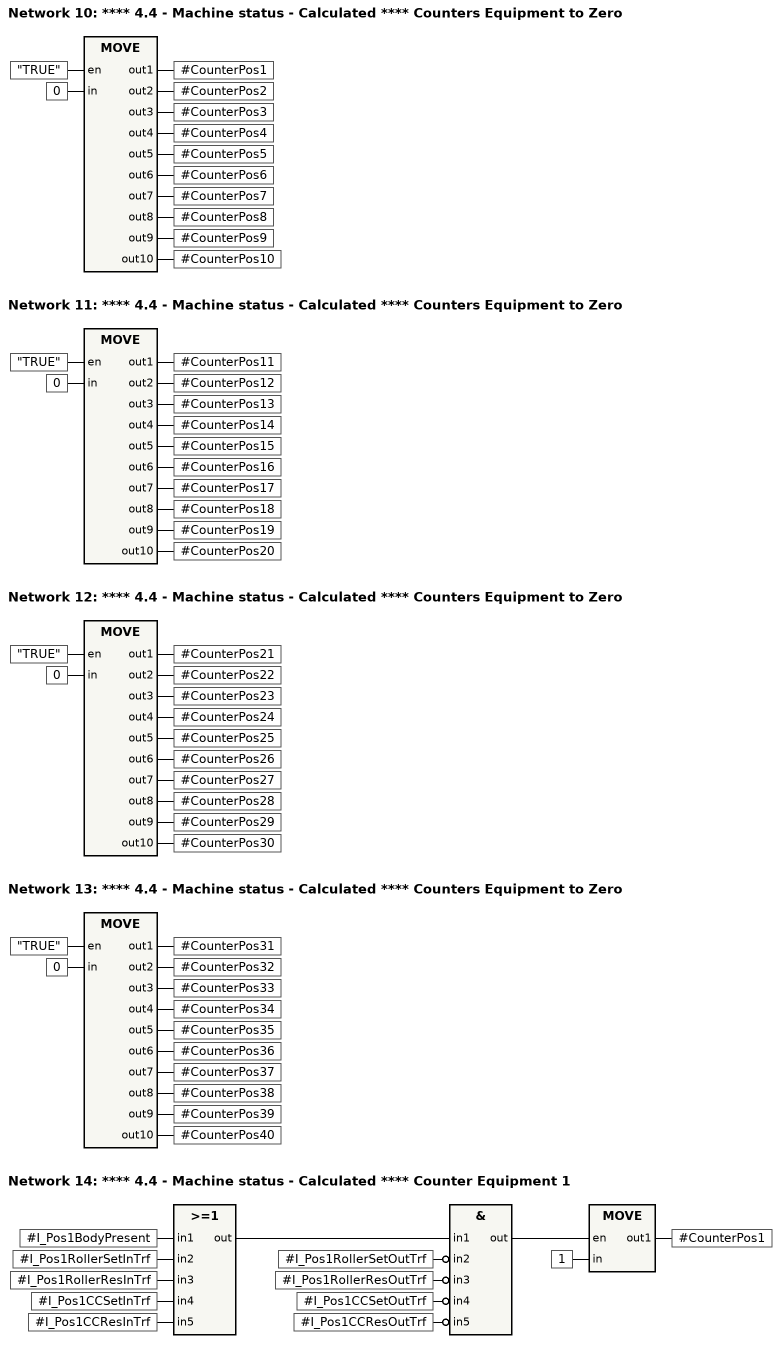
   IF "TRUE" THEN
       #CounterPos1 := 0;
       #CounterPos2 := 0;
       #CounterPos3 := 0;
       #CounterPos4 := 0;
       #CounterPos5 := 0;
       #CounterPos6 := 0;
       #CounterPos7 := 0;
       #CounterPos8 := 0;
       #CounterPos9 := 0;
       #CounterPos10 := 0;
   END_IF;
END_REGION

REGION Network 11: **** 4.4 - Machine status - Calculated **** Counters Equipment to Zero
   IF "TRUE" THEN
       #CounterPos11 := 0;
       #CounterPos12 := 0;
       #CounterPos13 := 0;
       #CounterPos14 := 0;
       #CounterPos15 := 0;
       #CounterPos16 := 0;
       #CounterPos17 := 0;
       #CounterPos18 := 0;
       #CounterPos19 := 0;
       #CounterPos20 := 0;
   END_IF;
END_REGION

REGION Network 12: **** 4.4 - Machine status - Calculated **** Counters Equipment to Zero
   IF "TRUE" THEN
       #CounterPos21 := 0;
       #CounterPos22 := 0;
       #CounterPos23 := 0;
       #CounterPos24 := 0;
       #CounterPos25 := 0;
       #CounterPos26 := 0;
       #CounterPos27 := 0;
       #CounterPos28 := 0;
       #CounterPos29 := 0;
       #CounterPos30 := 0;
   END_IF;
END_REGION

REGION Network 13: **** 4.4 - Machine status - Calculated **** Counters Equipment to Zero
   IF "TRUE" THEN
       #CounterPos31 := 0;
       #CounterPos32 := 0;
       #CounterPos33 := 0;
       #CounterPos34 := 0;
       #CounterPos35 := 0;
       #CounterPos36 := 0;
       #CounterPos37 := 0;
       #CounterPos38 := 0;
       #CounterPos39 := 0;
       #CounterPos40 := 0;
   END_IF;
END_REGION

REGION Network 14: **** 4.4 - Machine status - Calculated **** Counter Equipment 1
   IF (#I_Pos1BodyPresent OR #I_Pos1RollerSetInTrf OR #I_Pos1RollerResInTrf OR #I_Pos1CCSetInTrf OR #I_Pos1CCResInTrf) AND NOT #I_Pos1RollerSetOutTrf AND NOT #I_Pos1RollerResOutTrf AND NOT #I_Pos1CCSetOutTrf AND NOT #I_Pos1CCResOutTrf THEN
       #CounterPos1 := 1;
   END_IF;
END_REGION

REGION Network 15: **** 4.4 - Machine status - Calculated **** Counter Equipment 2
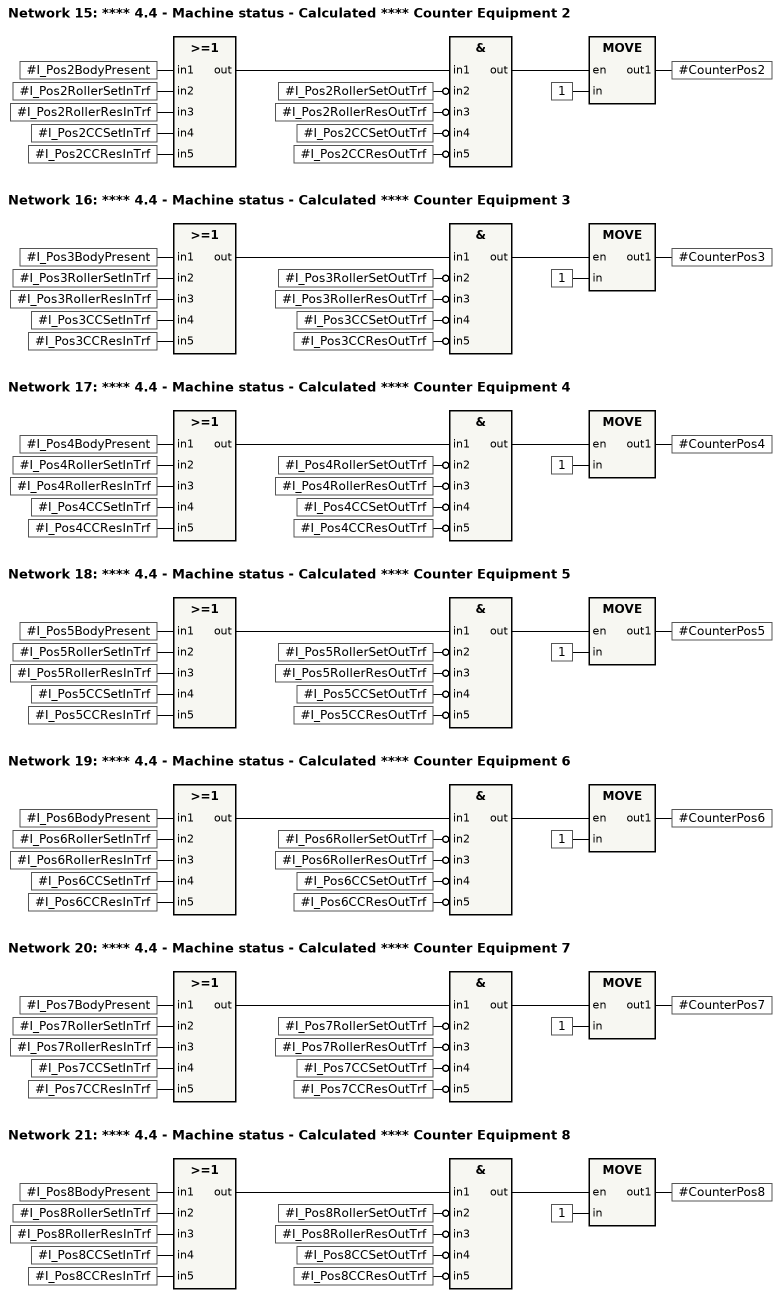
   IF (#I_Pos2BodyPresent OR #I_Pos2RollerSetInTrf OR #I_Pos2RollerResInTrf OR #I_Pos2CCSetInTrf OR #I_Pos2CCResInTrf) AND NOT #I_Pos2RollerSetOutTrf AND NOT #I_Pos2RollerResOutTrf AND NOT #I_Pos2CCSetOutTrf AND NOT #I_Pos2CCResOutTrf THEN
       #CounterPos2 := 1;
   END_IF;
END_REGION

REGION Network 16: **** 4.4 - Machine status - Calculated **** Counter Equipment 3
   IF (#I_Pos3BodyPresent OR #I_Pos3RollerSetInTrf OR #I_Pos3RollerResInTrf OR #I_Pos3CCSetInTrf OR #I_Pos3CCResInTrf) AND NOT #I_Pos3RollerSetOutTrf AND NOT #I_Pos3RollerResOutTrf AND NOT #I_Pos3CCSetOutTrf AND NOT #I_Pos3CCResOutTrf THEN
       #CounterPos3 := 1;
   END_IF;
END_REGION

REGION Network 17: **** 4.4 - Machine status - Calculated **** Counter Equipment 4
   IF (#I_Pos4BodyPresent OR #I_Pos4RollerSetInTrf OR #I_Pos4RollerResInTrf OR #I_Pos4CCSetInTrf OR #I_Pos4CCResInTrf) AND NOT #I_Pos4RollerSetOutTrf AND NOT #I_Pos4RollerResOutTrf AND NOT #I_Pos4CCSetOutTrf AND NOT #I_Pos4CCResOutTrf THEN
       #CounterPos4 := 1;
   END_IF;
END_REGION

REGION Network 18: **** 4.4 - Machine status - Calculated **** Counter Equipment 5
   IF (#I_Pos5BodyPresent OR #I_Pos5RollerSetInTrf OR #I_Pos5RollerResInTrf OR #I_Pos5CCSetInTrf OR #I_Pos5CCResInTrf) AND NOT #I_Pos5RollerSetOutTrf AND NOT #I_Pos5RollerResOutTrf AND NOT #I_Pos5CCSetOutTrf AND NOT #I_Pos5CCResOutTrf THEN
       #CounterPos5 := 1;
   END_IF;
END_REGION

REGION Network 19: **** 4.4 - Machine status - Calculated **** Counter Equipment 6
   IF (#I_Pos6BodyPresent OR #I_Pos6RollerSetInTrf OR #I_Pos6RollerResInTrf OR #I_Pos6CCSetInTrf OR #I_Pos6CCResInTrf) AND NOT #I_Pos6RollerSetOutTrf AND NOT #I_Pos6RollerResOutTrf AND NOT #I_Pos6CCSetOutTrf AND NOT #I_Pos6CCResOutTrf THEN
       #CounterPos6 := 1;
   END_IF;
END_REGION

REGION Network 20: **** 4.4 - Machine status - Calculated **** Counter Equipment 7
   IF (#I_Pos7BodyPresent OR #I_Pos7RollerSetInTrf OR #I_Pos7RollerResInTrf OR #I_Pos7CCSetInTrf OR #I_Pos7CCResInTrf) AND NOT #I_Pos7RollerSetOutTrf AND NOT #I_Pos7RollerResOutTrf AND NOT #I_Pos7CCSetOutTrf AND NOT #I_Pos7CCResOutTrf THEN
       #CounterPos7 := 1;
   END_IF;
END_REGION

REGION Network 21: **** 4.4 - Machine status - Calculated **** Counter Equipment 8
   IF (#I_Pos8BodyPresent OR #I_Pos8RollerSetInTrf OR #I_Pos8RollerResInTrf OR #I_Pos8CCSetInTrf OR #I_Pos8CCResInTrf) AND NOT #I_Pos8RollerSetOutTrf AND NOT #I_Pos8RollerResOutTrf AND NOT #I_Pos8CCSetOutTrf AND NOT #I_Pos8CCResOutTrf THEN
       #CounterPos8 := 1;
   END_IF;
END_REGION

REGION Network 22: **** 4.4 - Machine status - Calculated **** Counter Equipment 9
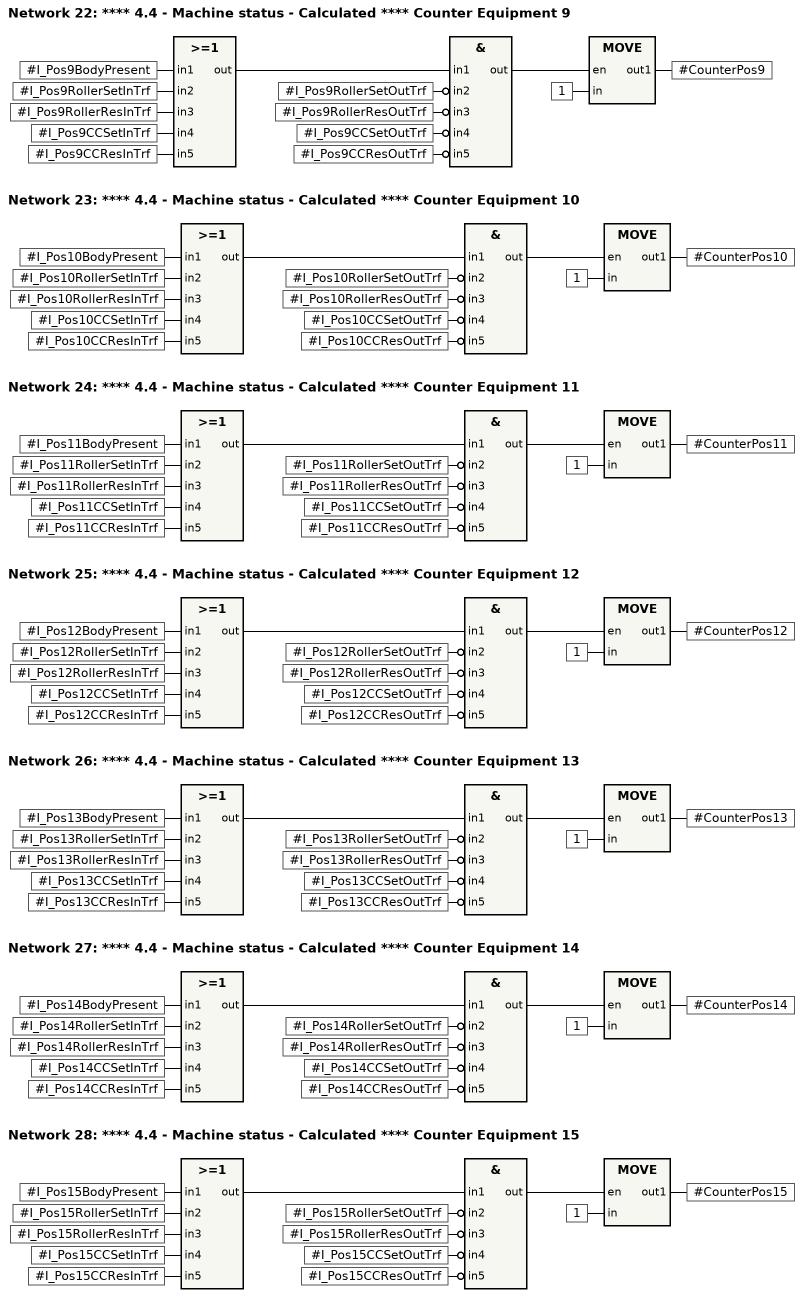
   IF (#I_Pos9BodyPresent OR #I_Pos9RollerSetInTrf OR #I_Pos9RollerResInTrf OR #I_Pos9CCSetInTrf OR #I_Pos9CCResInTrf) AND NOT #I_Pos9RollerSetOutTrf AND NOT #I_Pos9RollerResOutTrf AND NOT #I_Pos9CCSetOutTrf AND NOT #I_Pos9CCResOutTrf THEN
       #CounterPos9 := 1;
   END_IF;
END_REGION

REGION Network 23: **** 4.4 - Machine status - Calculated **** Counter Equipment 10
   IF (#I_Pos10BodyPresent OR #I_Pos10RollerSetInTrf OR #I_Pos10RollerResInTrf OR #I_Pos10CCSetInTrf OR #I_Pos10CCResInTrf) AND NOT #I_Pos10RollerSetOutTrf AND NOT #I_Pos10RollerResOutTrf AND NOT #I_Pos10CCSetOutTrf AND NOT #I_Pos10CCResOutTrf THEN
       #CounterPos10 := 1;
   END_IF;
END_REGION

REGION Network 24: **** 4.4 - Machine status - Calculated **** Counter Equipment 11
   IF (#I_Pos11BodyPresent OR #I_Pos11RollerSetInTrf OR #I_Pos11RollerResInTrf OR #I_Pos11CCSetInTrf OR #I_Pos11CCResInTrf) AND NOT #I_Pos11RollerSetOutTrf AND NOT #I_Pos11RollerResOutTrf AND NOT #I_Pos11CCSetOutTrf AND NOT #I_Pos11CCResOutTrf THEN
       #CounterPos11 := 1;
   END_IF;
END_REGION

REGION Network 25: **** 4.4 - Machine status - Calculated **** Counter Equipment 12
   IF (#I_Pos12BodyPresent OR #I_Pos12RollerSetInTrf OR #I_Pos12RollerResInTrf OR #I_Pos12CCSetInTrf OR #I_Pos12CCResInTrf) AND NOT #I_Pos12RollerSetOutTrf AND NOT #I_Pos12RollerResOutTrf AND NOT #I_Pos12CCSetOutTrf AND NOT #I_Pos12CCResOutTrf THEN
       #CounterPos12 := 1;
   END_IF;
END_REGION

REGION Network 26: **** 4.4 - Machine status - Calculated **** Counter Equipment 13
   IF (#I_Pos13BodyPresent OR #I_Pos13RollerSetInTrf OR #I_Pos13RollerResInTrf OR #I_Pos13CCSetInTrf OR #I_Pos13CCResInTrf) AND NOT #I_Pos13RollerSetOutTrf AND NOT #I_Pos13RollerResOutTrf AND NOT #I_Pos13CCSetOutTrf AND NOT #I_Pos13CCResOutTrf THEN
       #CounterPos13 := 1;
   END_IF;
END_REGION

REGION Network 27: **** 4.4 - Machine status - Calculated **** Counter Equipment 14
   IF (#I_Pos14BodyPresent OR #I_Pos14RollerSetInTrf OR #I_Pos14RollerResInTrf OR #I_Pos14CCSetInTrf OR #I_Pos14CCResInTrf) AND NOT #I_Pos14RollerSetOutTrf AND NOT #I_Pos14RollerResOutTrf AND NOT #I_Pos14CCSetOutTrf AND NOT #I_Pos14CCResOutTrf THEN
       #CounterPos14 := 1;
   END_IF;
END_REGION

REGION Network 28: **** 4.4 - Machine status - Calculated **** Counter Equipment 15
   IF (#I_Pos15BodyPresent OR #I_Pos15RollerSetInTrf OR #I_Pos15RollerResInTrf OR #I_Pos15CCSetInTrf OR #I_Pos15CCResInTrf) AND NOT #I_Pos15RollerSetOutTrf AND NOT #I_Pos15RollerResOutTrf AND NOT #I_Pos15CCSetOutTrf AND NOT #I_Pos15CCResOutTrf THEN
       #CounterPos15 := 1;
   END_IF;
END_REGION

REGION Network 29: **** 4.4 - Machine status - Calculated **** Counter Equipment 16
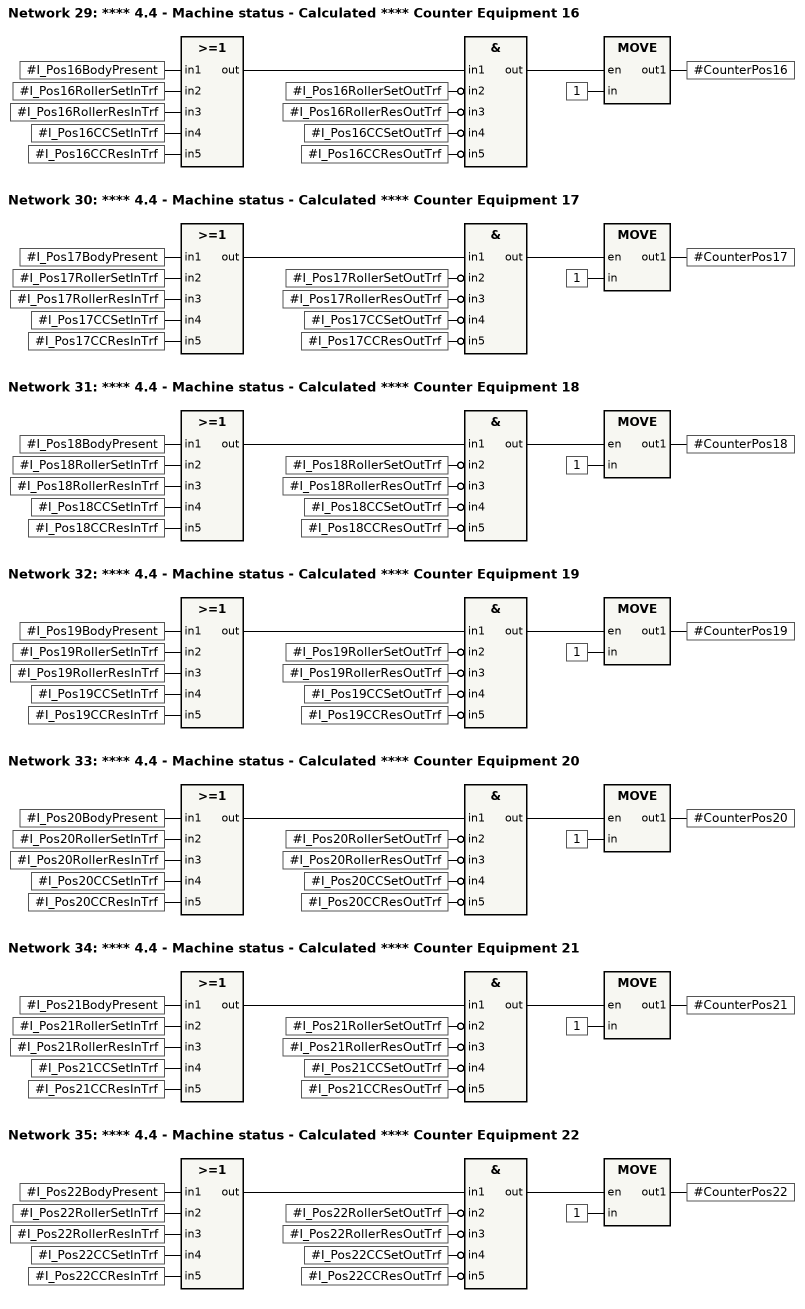
   IF (#I_Pos16BodyPresent OR #I_Pos16RollerSetInTrf OR #I_Pos16RollerResInTrf OR #I_Pos16CCSetInTrf OR #I_Pos16CCResInTrf) AND NOT #I_Pos16RollerSetOutTrf AND NOT #I_Pos16RollerResOutTrf AND NOT #I_Pos16CCSetOutTrf AND NOT #I_Pos16CCResOutTrf THEN
       #CounterPos16 := 1;
   END_IF;
END_REGION

REGION Network 30: **** 4.4 - Machine status - Calculated **** Counter Equipment 17
   IF (#I_Pos17BodyPresent OR #I_Pos17RollerSetInTrf OR #I_Pos17RollerResInTrf OR #I_Pos17CCSetInTrf OR #I_Pos17CCResInTrf) AND NOT #I_Pos17RollerSetOutTrf AND NOT #I_Pos17RollerResOutTrf AND NOT #I_Pos17CCSetOutTrf AND NOT #I_Pos17CCResOutTrf THEN
       #CounterPos17 := 1;
   END_IF;
END_REGION

REGION Network 31: **** 4.4 - Machine status - Calculated **** Counter Equipment 18
   IF (#I_Pos18BodyPresent OR #I_Pos18RollerSetInTrf OR #I_Pos18RollerResInTrf OR #I_Pos18CCSetInTrf OR #I_Pos18CCResInTrf) AND NOT #I_Pos18RollerSetOutTrf AND NOT #I_Pos18RollerResOutTrf AND NOT #I_Pos18CCSetOutTrf AND NOT #I_Pos18CCResOutTrf THEN
       #CounterPos18 := 1;
   END_IF;
END_REGION

REGION Network 32: **** 4.4 - Machine status - Calculated **** Counter Equipment 19
   IF (#I_Pos19BodyPresent OR #I_Pos19RollerSetInTrf OR #I_Pos19RollerResInTrf OR #I_Pos19CCSetInTrf OR #I_Pos19CCResInTrf) AND NOT #I_Pos19RollerSetOutTrf AND NOT #I_Pos19RollerResOutTrf AND NOT #I_Pos19CCSetOutTrf AND NOT #I_Pos19CCResOutTrf THEN
       #CounterPos19 := 1;
   END_IF;
END_REGION

REGION Network 33: **** 4.4 - Machine status - Calculated **** Counter Equipment 20
   IF (#I_Pos20BodyPresent OR #I_Pos20RollerSetInTrf OR #I_Pos20RollerResInTrf OR #I_Pos20CCSetInTrf OR #I_Pos20CCResInTrf) AND NOT #I_Pos20RollerSetOutTrf AND NOT #I_Pos20RollerResOutTrf AND NOT #I_Pos20CCSetOutTrf AND NOT #I_Pos20CCResOutTrf THEN
       #CounterPos20 := 1;
   END_IF;
END_REGION

REGION Network 34: **** 4.4 - Machine status - Calculated **** Counter Equipment 21
   IF (#I_Pos21BodyPresent OR #I_Pos21RollerSetInTrf OR #I_Pos21RollerResInTrf OR #I_Pos21CCSetInTrf OR #I_Pos21CCResInTrf) AND NOT #I_Pos21RollerSetOutTrf AND NOT #I_Pos21RollerResOutTrf AND NOT #I_Pos21CCSetOutTrf AND NOT #I_Pos21CCResOutTrf THEN
       #CounterPos21 := 1;
   END_IF;
END_REGION

REGION Network 35: **** 4.4 - Machine status - Calculated **** Counter Equipment 22
   IF (#I_Pos22BodyPresent OR #I_Pos22RollerSetInTrf OR #I_Pos22RollerResInTrf OR #I_Pos22CCSetInTrf OR #I_Pos22CCResInTrf) AND NOT #I_Pos22RollerSetOutTrf AND NOT #I_Pos22RollerResOutTrf AND NOT #I_Pos22CCSetOutTrf AND NOT #I_Pos22CCResOutTrf THEN
       #CounterPos22 := 1;
   END_IF;
END_REGION

REGION Network 36: **** 4.4 - Machine status - Calculated **** Counter Equipment 23
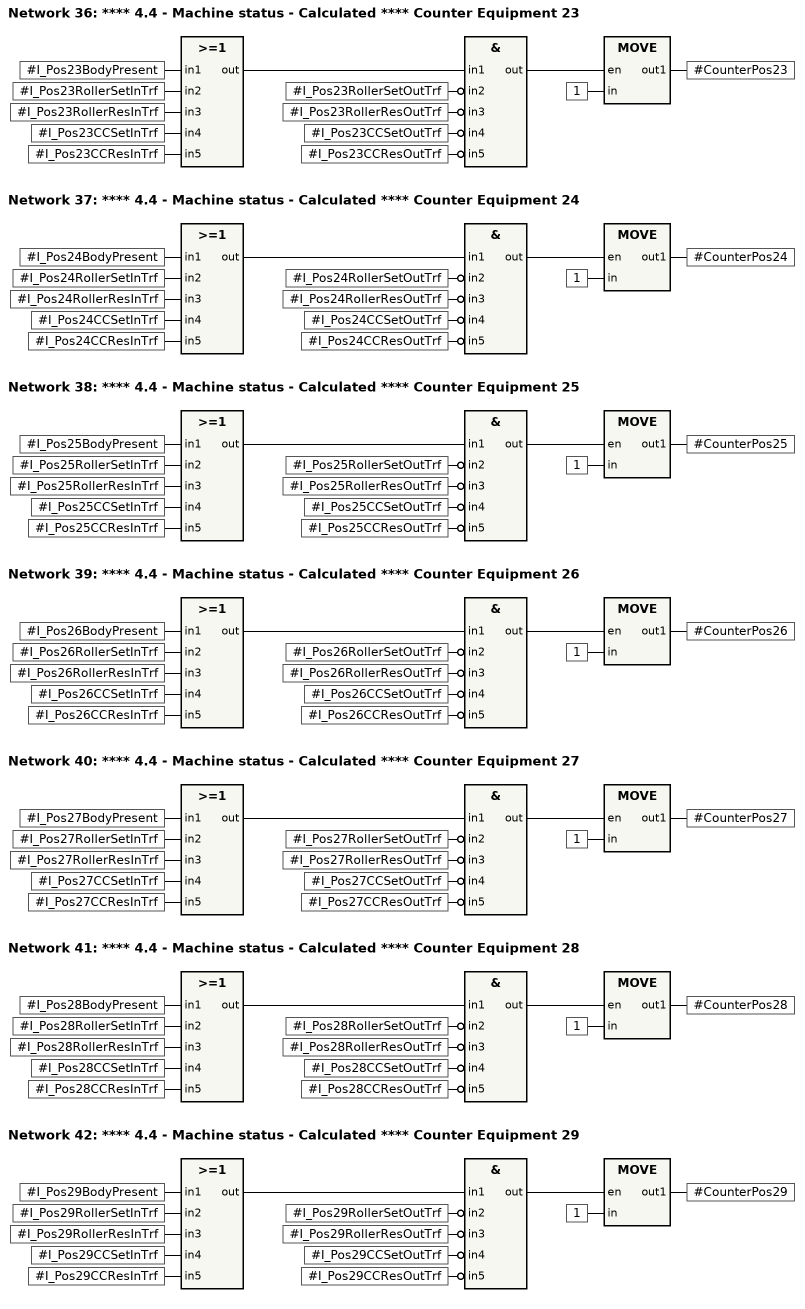
   IF (#I_Pos23BodyPresent OR #I_Pos23RollerSetInTrf OR #I_Pos23RollerResInTrf OR #I_Pos23CCSetInTrf OR #I_Pos23CCResInTrf) AND NOT #I_Pos23RollerSetOutTrf AND NOT #I_Pos23RollerResOutTrf AND NOT #I_Pos23CCSetOutTrf AND NOT #I_Pos23CCResOutTrf THEN
       #CounterPos23 := 1;
   END_IF;
END_REGION

REGION Network 37: **** 4.4 - Machine status - Calculated **** Counter Equipment 24
   IF (#I_Pos24BodyPresent OR #I_Pos24RollerSetInTrf OR #I_Pos24RollerResInTrf OR #I_Pos24CCSetInTrf OR #I_Pos24CCResInTrf) AND NOT #I_Pos24RollerSetOutTrf AND NOT #I_Pos24RollerResOutTrf AND NOT #I_Pos24CCSetOutTrf AND NOT #I_Pos24CCResOutTrf THEN
       #CounterPos24 := 1;
   END_IF;
END_REGION

REGION Network 38: **** 4.4 - Machine status - Calculated **** Counter Equipment 25
   IF (#I_Pos25BodyPresent OR #I_Pos25RollerSetInTrf OR #I_Pos25RollerResInTrf OR #I_Pos25CCSetInTrf OR #I_Pos25CCResInTrf) AND NOT #I_Pos25RollerSetOutTrf AND NOT #I_Pos25RollerResOutTrf AND NOT #I_Pos25CCSetOutTrf AND NOT #I_Pos25CCResOutTrf THEN
       #CounterPos25 := 1;
   END_IF;
END_REGION

REGION Network 39: **** 4.4 - Machine status - Calculated **** Counter Equipment 26
   IF (#I_Pos26BodyPresent OR #I_Pos26RollerSetInTrf OR #I_Pos26RollerResInTrf OR #I_Pos26CCSetInTrf OR #I_Pos26CCResInTrf) AND NOT #I_Pos26RollerSetOutTrf AND NOT #I_Pos26RollerResOutTrf AND NOT #I_Pos26CCSetOutTrf AND NOT #I_Pos26CCResOutTrf THEN
       #CounterPos26 := 1;
   END_IF;
END_REGION

REGION Network 40: **** 4.4 - Machine status - Calculated **** Counter Equipment 27
   IF (#I_Pos27BodyPresent OR #I_Pos27RollerSetInTrf OR #I_Pos27RollerResInTrf OR #I_Pos27CCSetInTrf OR #I_Pos27CCResInTrf) AND NOT #I_Pos27RollerSetOutTrf AND NOT #I_Pos27RollerResOutTrf AND NOT #I_Pos27CCSetOutTrf AND NOT #I_Pos27CCResOutTrf THEN
       #CounterPos27 := 1;
   END_IF;
END_REGION

REGION Network 41: **** 4.4 - Machine status - Calculated **** Counter Equipment 28
   IF (#I_Pos28BodyPresent OR #I_Pos28RollerSetInTrf OR #I_Pos28RollerResInTrf OR #I_Pos28CCSetInTrf OR #I_Pos28CCResInTrf) AND NOT #I_Pos28RollerSetOutTrf AND NOT #I_Pos28RollerResOutTrf AND NOT #I_Pos28CCSetOutTrf AND NOT #I_Pos28CCResOutTrf THEN
       #CounterPos28 := 1;
   END_IF;
END_REGION

REGION Network 42: **** 4.4 - Machine status - Calculated **** Counter Equipment 29
   IF (#I_Pos29BodyPresent OR #I_Pos29RollerSetInTrf OR #I_Pos29RollerResInTrf OR #I_Pos29CCSetInTrf OR #I_Pos29CCResInTrf) AND NOT #I_Pos29RollerSetOutTrf AND NOT #I_Pos29RollerResOutTrf AND NOT #I_Pos29CCSetOutTrf AND NOT #I_Pos29CCResOutTrf THEN
       #CounterPos29 := 1;
   END_IF;
END_REGION

REGION Network 43: **** 4.4 - Machine status - Calculated **** Counter Equipment 30
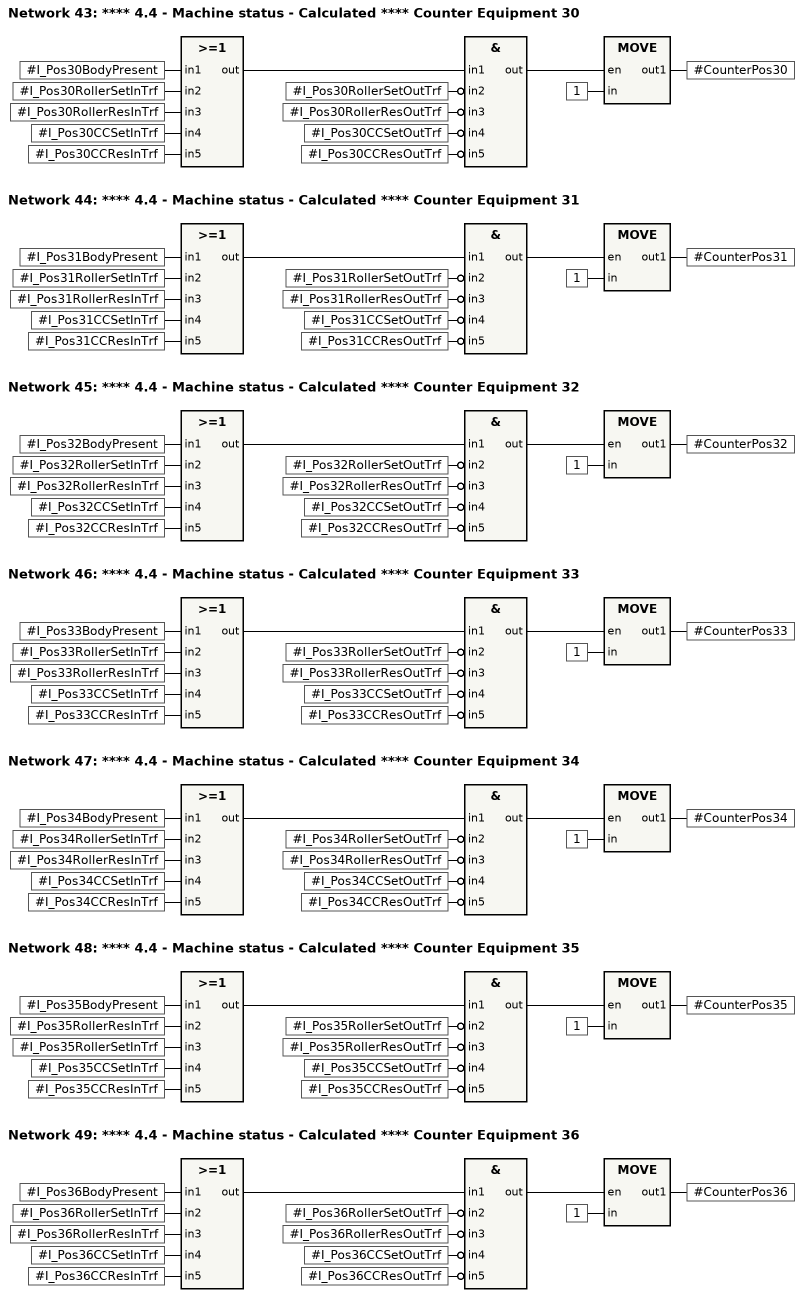
   IF (#I_Pos30BodyPresent OR #I_Pos30RollerSetInTrf OR #I_Pos30RollerResInTrf OR #I_Pos30CCSetInTrf OR #I_Pos30CCResInTrf) AND NOT #I_Pos30RollerSetOutTrf AND NOT #I_Pos30RollerResOutTrf AND NOT #I_Pos30CCSetOutTrf AND NOT #I_Pos30CCResOutTrf THEN
       #CounterPos30 := 1;
   END_IF;
END_REGION

REGION Network 44: **** 4.4 - Machine status - Calculated **** Counter Equipment 31
   IF (#I_Pos31BodyPresent OR #I_Pos31RollerSetInTrf OR #I_Pos31RollerResInTrf OR #I_Pos31CCSetInTrf OR #I_Pos31CCResInTrf) AND NOT #I_Pos31RollerSetOutTrf AND NOT #I_Pos31RollerResOutTrf AND NOT #I_Pos31CCSetOutTrf AND NOT #I_Pos31CCResOutTrf THEN
       #CounterPos31 := 1;
   END_IF;
END_REGION

REGION Network 45: **** 4.4 - Machine status - Calculated **** Counter Equipment 32
   IF (#I_Pos32BodyPresent OR #I_Pos32RollerSetInTrf OR #I_Pos32RollerResInTrf OR #I_Pos32CCSetInTrf OR #I_Pos32CCResInTrf) AND NOT #I_Pos32RollerSetOutTrf AND NOT #I_Pos32RollerResOutTrf AND NOT #I_Pos32CCSetOutTrf AND NOT #I_Pos32CCResOutTrf THEN
       #CounterPos32 := 1;
   END_IF;
END_REGION

REGION Network 46: **** 4.4 - Machine status - Calculated **** Counter Equipment 33
   IF (#I_Pos33BodyPresent OR #I_Pos33RollerSetInTrf OR #I_Pos33RollerResInTrf OR #I_Pos33CCSetInTrf OR #I_Pos33CCResInTrf) AND NOT #I_Pos33RollerSetOutTrf AND NOT #I_Pos33RollerResOutTrf AND NOT #I_Pos33CCSetOutTrf AND NOT #I_Pos33CCResOutTrf THEN
       #CounterPos33 := 1;
   END_IF;
END_REGION

REGION Network 47: **** 4.4 - Machine status - Calculated **** Counter Equipment 34
   IF (#I_Pos34BodyPresent OR #I_Pos34RollerSetInTrf OR #I_Pos34RollerResInTrf OR #I_Pos34CCSetInTrf OR #I_Pos34CCResInTrf) AND NOT #I_Pos34RollerSetOutTrf AND NOT #I_Pos34RollerResOutTrf AND NOT #I_Pos34CCSetOutTrf AND NOT #I_Pos34CCResOutTrf THEN
       #CounterPos34 := 1;
   END_IF;
END_REGION

REGION Network 48: **** 4.4 - Machine status - Calculated **** Counter Equipment 35
   IF (#I_Pos35BodyPresent OR #I_Pos35RollerResInTrf OR #I_Pos35RollerSetInTrf OR #I_Pos35CCSetInTrf OR #I_Pos35CCResInTrf) AND NOT #I_Pos35RollerSetOutTrf AND NOT #I_Pos35RollerResOutTrf AND NOT #I_Pos35CCSetOutTrf AND NOT #I_Pos35CCResOutTrf THEN
       #CounterPos35 := 1;
   END_IF;
END_REGION

REGION Network 49: **** 4.4 - Machine status - Calculated **** Counter Equipment 36
   IF (#I_Pos36BodyPresent OR #I_Pos36RollerSetInTrf OR #I_Pos36RollerResInTrf OR #I_Pos36CCSetInTrf OR #I_Pos36CCResInTrf) AND NOT #I_Pos36RollerSetOutTrf AND NOT #I_Pos36RollerResOutTrf AND NOT #I_Pos36CCSetOutTrf AND NOT #I_Pos36CCResOutTrf THEN
       #CounterPos36 := 1;
   END_IF;
END_REGION

REGION Network 50: **** 4.4 - Machine status - Calculated **** Counter Equipment 37
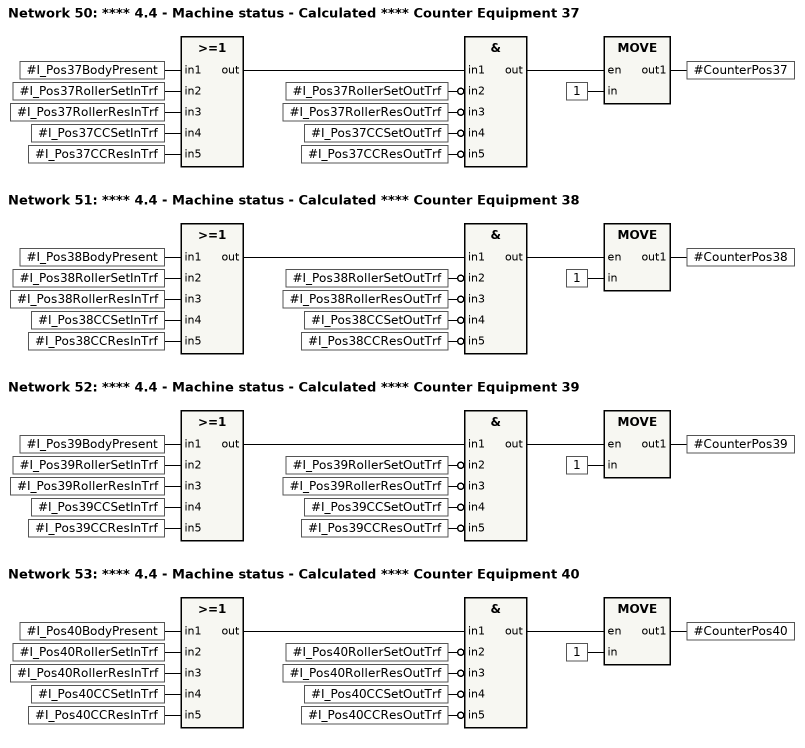
   IF (#I_Pos37BodyPresent OR #I_Pos37RollerSetInTrf OR #I_Pos37RollerResInTrf OR #I_Pos37CCSetInTrf OR #I_Pos37CCResInTrf) AND NOT #I_Pos37RollerSetOutTrf AND NOT #I_Pos37RollerResOutTrf AND NOT #I_Pos37CCSetOutTrf AND NOT #I_Pos37CCResOutTrf THEN
       #CounterPos37 := 1;
   END_IF;
END_REGION

REGION Network 51: **** 4.4 - Machine status - Calculated **** Counter Equipment 38
   IF (#I_Pos38BodyPresent OR #I_Pos38RollerSetInTrf OR #I_Pos38RollerResInTrf OR #I_Pos38CCSetInTrf OR #I_Pos38CCResInTrf) AND NOT #I_Pos38RollerSetOutTrf AND NOT #I_Pos38RollerResOutTrf AND NOT #I_Pos38CCSetOutTrf AND NOT #I_Pos38CCResOutTrf THEN
       #CounterPos38 := 1;
   END_IF;
END_REGION

REGION Network 52: **** 4.4 - Machine status - Calculated **** Counter Equipment 39
   IF (#I_Pos39BodyPresent OR #I_Pos39RollerSetInTrf OR #I_Pos39RollerResInTrf OR #I_Pos39CCSetInTrf OR #I_Pos39CCResInTrf) AND NOT #I_Pos39RollerSetOutTrf AND NOT #I_Pos39RollerResOutTrf AND NOT #I_Pos39CCSetOutTrf AND NOT #I_Pos39CCResOutTrf THEN
       #CounterPos39 := 1;
   END_IF;
END_REGION

REGION Network 53: **** 4.4 - Machine status - Calculated **** Counter Equipment 40
   IF (#I_Pos40BodyPresent OR #I_Pos40RollerSetInTrf OR #I_Pos40RollerResInTrf OR #I_Pos40CCSetInTrf OR #I_Pos40CCResInTrf) AND NOT #I_Pos40RollerSetOutTrf AND NOT #I_Pos40RollerResOutTrf AND NOT #I_Pos40CCSetOutTrf AND NOT #I_Pos40CCResOutTrf THEN
       #CounterPos40 := 1;
   END_IF;
END_REGION

REGION Network 54: **** 4.4 - Machine status - Calculated **** Writing the Counter Value
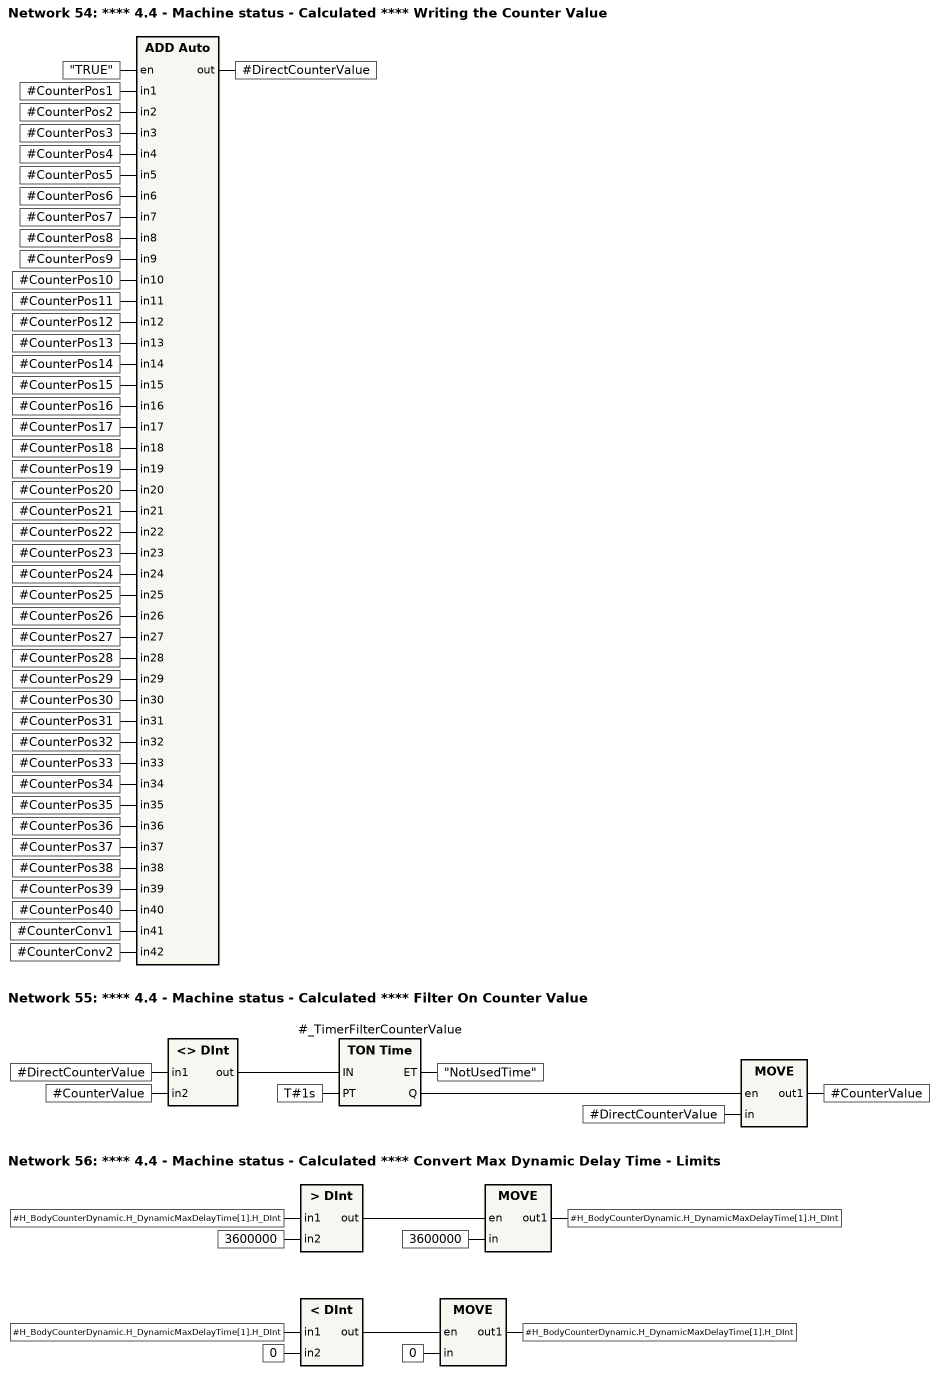
   IF "TRUE" THEN
       #DirectCounterValue := #CounterPos1 + #CounterPos2 + #CounterPos3 + #CounterPos4 + #CounterPos5 + #CounterPos6 + #CounterPos7 + #CounterPos8 + #CounterPos9 + #CounterPos10 + #CounterPos11 + #CounterPos12 + #CounterPos13 + #CounterPos14 + #CounterPos15 + #CounterPos16 + #CounterPos17 + #CounterPos18 + #CounterPos19 + #CounterPos20 + #CounterPos21 + #CounterPos22 + #CounterPos23 + #CounterPos24 + #CounterPos25 + #CounterPos26 + #CounterPos27 + #CounterPos28 + #CounterPos29 + #CounterPos30 + #CounterPos31 + #CounterPos32 + #CounterPos33 + #CounterPos34 + #CounterPos35 + #CounterPos36 + #CounterPos37 + #CounterPos38 + #CounterPos39 + #CounterPos40 + #CounterConv1 + #CounterConv2;
   END_IF;
END_REGION

REGION Network 55: **** 4.4 - Machine status - Calculated **** Filter On Counter Value
   #_TimerFilterCounterValue(IN := #DirectCounterValue <> #CounterValue, PT := T#1s, ET => "NotUsedTime");   // TON
   IF #_TimerFilterCounterValue.Q THEN #CounterValue := #DirectCounterValue; END_IF;
END_REGION

REGION Network 56: **** 4.4 - Machine status - Calculated **** Convert Max Dynamic Delay Time - Limits
   IF #H_BodyCounterDynamic.H_DynamicMaxDelayTime[1].H_DInt > 3600000 THEN
       #H_BodyCounterDynamic.H_DynamicMaxDelayTime[1].H_DInt := 3600000;
   END_IF;
   IF #H_BodyCounterDynamic.H_DynamicMaxDelayTime[1].H_DInt < 0 THEN
       #H_BodyCounterDynamic.H_DynamicMaxDelayTime[1].H_DInt := 0;
   END_IF;
END_REGION

REGION Network 57: **** 4.4 - Machine status - Calculated **** Convert Max Dynamic Delay Time
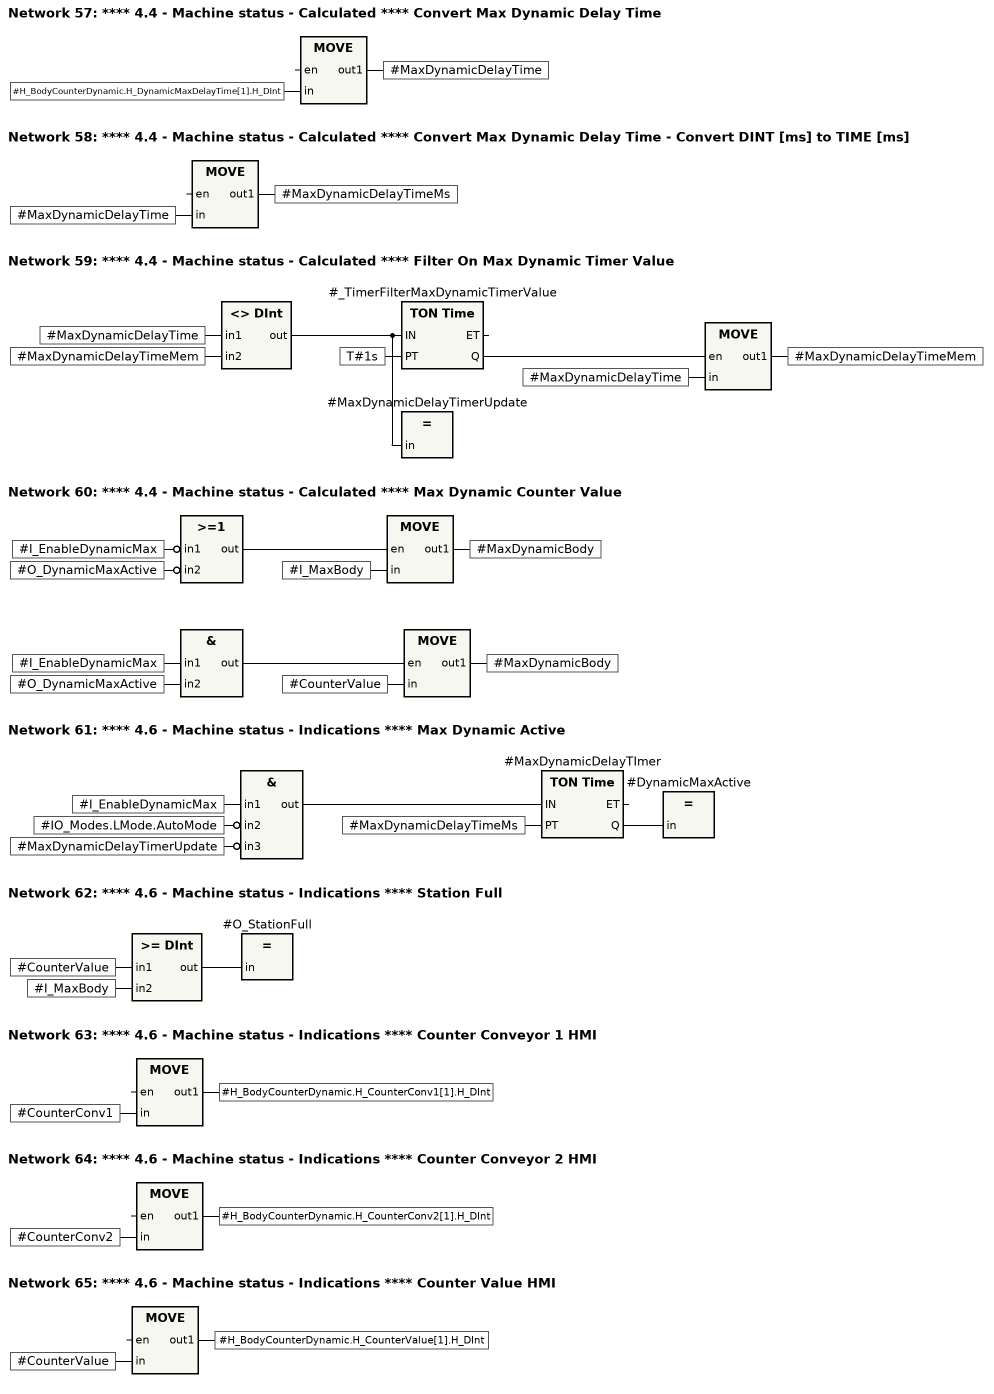
   #MaxDynamicDelayTime := #H_BodyCounterDynamic.H_DynamicMaxDelayTime[1].H_DInt;
END_REGION

REGION Network 58: **** 4.4 - Machine status - Calculated **** Convert Max Dynamic Delay Time - Convert DINT [ms] to TIME [ms]
   #MaxDynamicDelayTimeMs := #MaxDynamicDelayTime;
END_REGION

REGION Network 59: **** 4.4 - Machine status - Calculated **** Filter On Max Dynamic Timer Value
   #_w1 := #MaxDynamicDelayTime <> #MaxDynamicDelayTimeMem;
   #_TimerFilterMaxDynamicTimerValue(IN := #_w1, PT := T#1s);   // TON
   IF #_TimerFilterMaxDynamicTimerValue.Q THEN #MaxDynamicDelayTimeMem := #MaxDynamicDelayTime; END_IF;
   #MaxDynamicDelayTimerUpdate := #_w1;
END_REGION

REGION Network 60: **** 4.4 - Machine status - Calculated **** Max Dynamic Counter Value
   IF NOT #I_EnableDynamicMax OR NOT #O_DynamicMaxActive THEN #MaxDynamicBody := #I_MaxBody; END_IF;
   IF #I_EnableDynamicMax AND #O_DynamicMaxActive THEN #MaxDynamicBody := #CounterValue; END_IF;
END_REGION

REGION Network 61: **** 4.6 - Machine status - Indications **** Max Dynamic Active
   #MaxDynamicDelayTImer(IN := #I_EnableDynamicMax AND NOT #IO_Modes.LMode.AutoMode AND NOT #MaxDynamicDelayTimerUpdate,   // TON
                         PT := #MaxDynamicDelayTimeMs);
   #DynamicMaxActive := #MaxDynamicDelayTImer.Q;
END_REGION

REGION Network 62: **** 4.6 - Machine status - Indications **** Station Full
   #O_StationFull := #CounterValue >= #I_MaxBody;
END_REGION

REGION Network 63: **** 4.6 - Machine status - Indications **** Counter Conveyor 1 HMI
   #H_BodyCounterDynamic.H_CounterConv1[1].H_DInt := #CounterConv1;
END_REGION

REGION Network 64: **** 4.6 - Machine status - Indications **** Counter Conveyor 2 HMI
   #H_BodyCounterDynamic.H_CounterConv2[1].H_DInt := #CounterConv2;
END_REGION

REGION Network 65: **** 4.6 - Machine status - Indications **** Counter Value HMI
   #H_BodyCounterDynamic.H_CounterValue[1].H_DInt := #CounterValue;
END_REGION

REGION Network 66: **** 4.6 - Machine status - Indications **** Dynamic Max Delay Time Value HMI
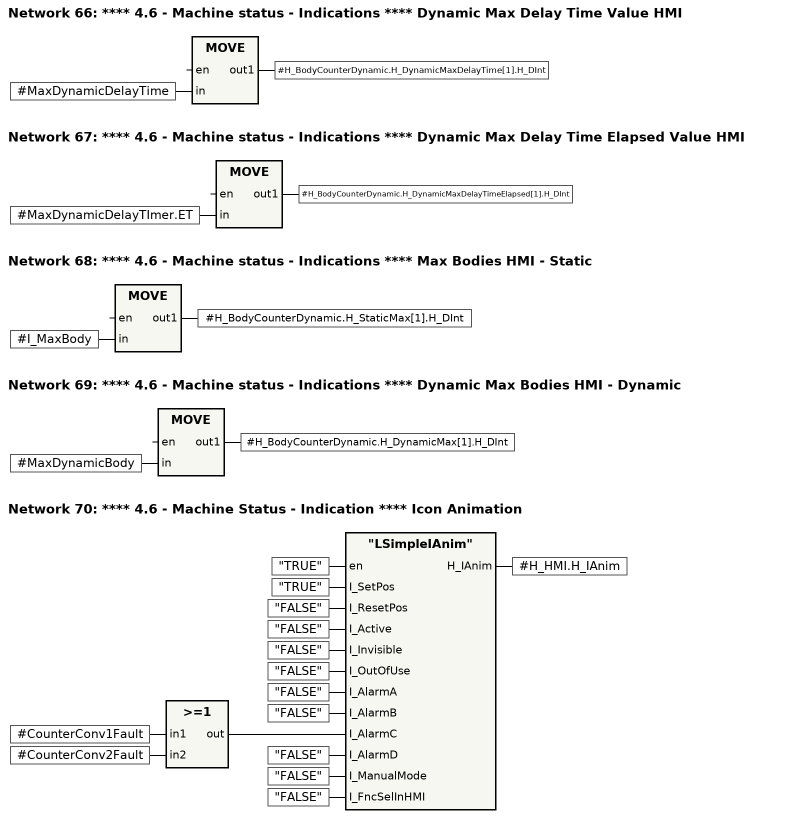
   #H_BodyCounterDynamic.H_DynamicMaxDelayTime[1].H_DInt := #MaxDynamicDelayTime;
END_REGION

REGION Network 67: **** 4.6 - Machine status - Indications **** Dynamic Max Delay Time Elapsed Value HMI
   #H_BodyCounterDynamic.H_DynamicMaxDelayTimeElapsed[1].H_DInt := #MaxDynamicDelayTImer.ET;
END_REGION

